LIN {X 0,Y 373.397,Z 455.176,A -85,B 0,C 180,E1 -12866.615,E2 -12866.615} C_VEL
LIN {X 0,Y 372.645,Z 466.782,A -85,B 0,C 180,E1 -12867.431,E2 -12867.431} C_VEL
LIN {X 0,Y 371.772,Z 478.488,A -85,B 0,C 180,E1 -12868.51,E2 -12868.51} C_VEL
LIN {X 0,Y 370.845,Z 489.006,A -85,B 0,C 180,E1 -12869.728,E2 -12869.728} C_VEL
LIN {X 0,Y 369.997,Z 498.484,A -85,B 0,C 180,E1 -12871.087,E2 -12871.087} C_VEL
LIN {X 0,Y 369.105,Z 507.613,A -85,B 0,C 180,E1 -12872.727,E2 -12872.727} C_VEL
LIN {X 0,Y 368.474,Z 514.962,A -85,B 0,C 180,E1 -12874.374,E2 -12874.374} C_VEL
LIN {X 0,Y 368.116,Z 520.845,A -85,B 0,C 180,E1 -12876.026,E2 -12876.026} C_VEL
LIN {X 0,Y 367.769,Z 525.5,A -85,B 0,C 180,E1 -12877.686,E2 -12877.686} C_VEL
LIN {X 0,Y 367.515,Z 529.046,A -85,B 0,C 180,E1 -12879.354,E2 -12879.354} C_VEL
LIN {X 0,Y 367.376,Z 531.568,A -85,B 0,C 180,E1 -12881.028,E2 -12881.028} C_VEL
LIN {X 0,Y 367.353,Z 533.088,A -85,B 0,C 180,E1 -12882.657,E2 -12882.657} C_VEL
LIN {X 0,Y 367.241,Z 533.754,A -85,B 0,C 180,E1 -12884.404,E2 -12884.404} C_VEL
LIN {X 0,Y 367.257,Z 533.671,A -85,B 0,C 180,E1 -12885.539,E2 -12885.539} C_VEL
LIN {X 0,Y 367.386,Z 532.771,A -85,B 0,C 180,E1 -12887.131,E2 -12887.131} C_VEL
LIN {X 0,Y 367.617,Z 530.783,A -85,B 0,C 180,E1 -12888.964,E2 -12888.964} C_VEL
LIN {X 0,Y 367.953,Z 527.938,A -85,B 0,C 180,E1 -12890.625,E2 -12890.625} C_VEL
LIN {X 0,Y 368.238,Z 525.407,A -85,B 0,C 180,E1 -12891.755,E2 -12891.755} C_VEL
LIN {X 0,Y 367.828,Z 523.313,A -85,B 0,C 180,E1 -12892.614,E2 -12892.614} C_VEL
LIN {X 0,Y 365.519,Z 519.519,A -85,B 0,C 180,E1 -12894.001,E2 -12894.001} C_VEL
LIN {X 0,Y 363.313,Z 515.047,A -85,B 0,C 180,E1 -12895.351,E2 -12895.351} C_VEL
LIN {X 0,Y 363.065,Z 511.888,A -85,B 0,C 180,E1 -12896.139,E2 -12896.139} C_VEL
LIN {X 0,Y 364.268,Z 503.365,A -85,B 0,C 180,E1 -12897.895,E2 -12897.895} C_VEL
LIN {X 0,Y 365.394,Z 494.439,A -85,B 0,C 180,E1 -12899.37,E2 -12899.37} C_VEL
LIN {X 0,Y 366.725,Z 483.898,A -85,B 0,C 180,E1 -12900.759,E2 -12900.759} C_VEL
LIN {X 0,Y 367.92,Z 473.579,A -85,B 0,C 180,E1 -12901.848,E2 -12901.848} C_VEL
LIN {X 0,Y 368.964,Z 462.928,A -85,B 0,C 180,E1 -12902.747,E2 -12902.747} C_VEL
LIN {X 0,Y 369.916,Z 451.086,A -85,B 0,C 180,E1 -12903.514,E2 -12903.514} C_VEL
LIN {X 0,Y 370.609,Z 438.576,A -85,B 0,C 180,E1 -12904.096,E2 -12904.096} C_VEL
LIN {X 0,Y 371.139,Z 424.92,A -85,B 0,C 180,E1 -12904.492,E2 -12904.492} C_VEL
LIN {X 0,Y 372.654,Z 349.861,A -85,B 0,C 180,E1 -12905.968,E2 -12905.968} C_VEL
LIN {X 0,Y 368.76,Z 332.715,A -85,B 0,C 180,E1 -12906.629,E2 -12906.629} C_VEL
LIN {X 0,Y 364.625,Z 322.839,A -85,B 0,C 180,E1 -12907.207,E2 -12907.207} C_VEL
LIN {X 0,Y 362.63,Z 313.77,A -85,B 0,C 180,E1 -12909.757,E2 -12909.757} C_VEL
LIN {X 0,Y 361.806,Z 310.419,A -85,B 0,C 180,E1 -12910.75,E2 -12910.75} C_VEL
LIN {X 0,Y 361.809,Z 310.418,A -85,B 0,C 180,E1 -12914.368,E2 -12914.368} C_VEL
LIN {X 0,Y 361.822,Z 310.407,A -85,B 0,C 180,E1 -12917.569,E2 -12917.569} C_VEL
LIN {X 0,Y 361.836,Z 310.414,A -85,B 0,C 180,E1 -12921.572,E2 -12921.572} C_VEL
LIN {X 0,Y 361.865,Z 310.406,A -85,B 0,C 180,E1 -12924.655,E2 -12924.655} C_VEL
LIN {X 0,Y 361.829,Z 310.412,A -85,B 0,C 180,E1 -12928.37,E2 -12928.37} C_VEL
LIN {X 0,Y 361.857,Z 310.404,A -85,B 0,C 180,E1 -12930.952,E2 -12930.952} C_VEL
LIN {X 0,Y 361.859,Z 310.405,A -85,B 0,C 180,E1 -12934.705,E2 -12934.705} C_VEL
LIN {X 0,Y 361.852,Z 310.407,A -85,B 0,C 180,E1 -12938.345,E2 -12938.345} C_VEL
LIN {X 0,Y 361.895,Z 310.399,A -85,B 0,C 180,E1 -12942.093,E2 -12942.093} C_VEL
LIN {X 0,Y 361.97,Z 310.388,A -85,B 0,C 180,E1 -12946.113,E2 -12946.113} C_VEL
LIN {X 0,Y 361.985,Z 310.393,A -85,B 0,C 180,E1 -12949.937,E2 -12949.937} C_VEL
LIN {X 0,Y 362.106,Z 310.375,A -85,B 0,C 180,E1 -12953.313,E2 -12953.313} C_VEL
LIN {X 0,Y 362.246,Z 310.353,A -85,B 0,C 180,E1 -12957.776,E2 -12957.776} C_VEL
LIN {X 0,Y 362.247,Z 310.351,A -85,B 0,C 180,E1 -12962.224,E2 -12962.224} C_VEL
LIN {X 0,Y 362.131,Z 310.368,A -85,B 0,C 180,E1 -12966.687,E2 -12966.687} C_VEL
LIN {X 0,Y 361.988,Z 310.389,A -85,B 0,C 180,E1 -12970.064,E2 -12970.064} C_VEL
LIN {X 0,Y 361.99,Z 310.382,A -85,B 0,C 180,E1 -12973.899,E2 -12973.899} C_VEL
LIN {X 0,Y 361.92,Z 310.396,A -85,B 0,C 180,E1 -12976.935,E2 -12976.935} C_VEL
LIN {X 0,Y 361.879,Z 310.403,A -85,B 0,C 180,E1 -12980.462,E2 -12980.462} C_VEL
LIN {X 0,Y 361.853,Z 310.405,A -85,B 0,C 180,E1 -12984.102,E2 -12984.102} C_VEL
LIN {X 0,Y 361.838,Z 310.406,A -85,B 0,C 180,E1 -12987.785,E2 -12987.785} C_VEL
LIN {X 0,Y 361.84,Z 310.408,A -85,B 0,C 180,E1 -12991.286,E2 -12991.286} C_VEL
LIN {X 0,Y 361.848,Z 310.409,A -85,B 0,C 180,E1 -12994.281,E2 -12994.281} C_VEL
LIN {X 0,Y 361.854,Z 310.411,A -85,B 0,C 180,E1 -12997.223,E2 -12997.223} C_VEL
LIN {X 0,Y 361.807,Z 310.416,A -85,B 0,C 180,E1 -13000.752,E2 -13000.752} C_VEL
LIN {X 0,Y 361.811,Z 310.405,A -85,B 0,C 180,E1 -13004.37,E2 -13004.37} C_VEL
LIN {X 0,Y 361.831,Z 310.415,A -85,B 0,C 180,E1 -13007.569,E2 -13007.569} C_VEL
LIN {X 0,Y 361.862,Z 310.412,A -85,B 0,C 180,E1 -13010.975,E2 -13010.975} C_VEL
LIN {X 0,Y 361.871,Z 310.406,A -85,B 0,C 180,E1 -13014.656,E2 -13014.656} C_VEL
LIN {X 0,Y 361.835,Z 310.411,A -85,B 0,C 180,E1 -13018.372,E2 -13018.372} C_VEL
LIN {X 0,Y 361.903,Z 310.527,A -85,B 0,C 180,E1 -13019.004,E2 -13019.004} C_VEL
LIN {X 0,Y 364.589,Z 321.736,A -85,B 0,C 180,E1 -13022.133,E2 -13022.133} C_VEL
LIN {X 0,Y 366.327,Z 331.239,A -85,B 0,C 180,E1 -13024.628,E2 -13024.628} C_VEL
LIN {X 0,Y 366.472,Z 334.158,A -85,B 0,C 180,E1 -13025.349,E2 -13025.349} C_VEL
LIN {X 0,Y 365.703,Z 341.412,A -85,B 0,C 180,E1 -13026.981,E2 -13026.981} C_VEL
LIN {X 0,Y 370.351,Z 363.93,A -85,B 0,C 180,E1 -13027.82,E2 -13027.82} C_VEL
LIN {X 0,Y 372.213,Z 375.715,A -85,B 0,C 180,E1 -13028.207,E2 -13028.207} C_VEL
LIN {X 0,Y 370.773,Z 449.685,A -85,B 0,C 180,E1 -13029.69,E2 -13029.69} C_VEL
LIN {X 0,Y 369.999,Z 462.791,A -85,B 0,C 180,E1 -13030.153,E2 -13030.153} C_VEL
LIN {X 0,Y 369.057,Z 475.405,A -85,B 0,C 180,E1 -13030.824,E2 -13030.824} C_VEL
LIN {X 0,Y 367.953,Z 486.664,A -85,B 0,C 180,E1 -13031.631,E2 -13031.631} C_VEL
LIN {X 0,Y 366.614,Z 498.29,A -85,B 0,C 180,E1 -13032.716,E2 -13032.716} C_VEL
LIN {X 0,Y 365.281,Z 508.754,A -85,B 0,C 180,E1 -13033.945,E2 -13033.945} C_VEL
LIN {X 0,Y 364.256,Z 517.807,A -85,B 0,C 180,E1 -13035.268,E2 -13035.268} C_VEL
LIN {X 0,Y 363.039,Z 526.654,A -85,B 0,C 180,E1 -13036.853,E2 -13036.853} C_VEL
LIN {X 0,Y 362.012,Z 534.145,A -85,B 0,C 180,E1 -13038.523,E2 -13038.523} C_VEL
LIN {X 0,Y 361.207,Z 541.091,A -85,B 0,C 180,E1 -13040.482,E2 -13040.482} C_VEL
LIN {X 0,Y 360.731,Z 545.697,A -85,B 0,C 180,E1 -13042.163,E2 -13042.163} C_VEL
LIN {X 0,Y 360.425,Z 549.441,A -85,B 0,C 180,E1 -13043.969,E2 -13043.969} C_VEL
LIN {X 0,Y 360.349,Z 551.741,A -85,B 0,C 180,E1 -13045.527,E2 -13045.527} C_VEL
LIN {X 0,Y 360.296,Z 552.926,A -85,B 0,C 180,E1 -13046.646,E2 -13046.646} C_VEL
LIN {X 0,Y 360.303,Z 554.036,A -85,B 0,C 180,E1 -13048.883,E2 -13048.883} C_VEL
LIN {X 0,Y 360.36,Z 554.014,A -85,B 0,C 180,E1 -13050.001,E2 -13050.001} C_VEL
LIN {X 0,Y 360.321,Z 553.599,A -85,B 0,C 180,E1 -13051.119,E2 -13051.119} C_VEL
LIN {X 0,Y 360.279,Z 552.743,A -85,B 0,C 180,E1 -13052.237,E2 -13052.237} C_VEL
LIN {X 0,Y 360.303,Z 551.485,A -85,B 0,C 180,E1 -13053.356,E2 -13053.356} C_VEL
LIN {X 0,Y 360.368,Z 548.805,A -85,B 0,C 180,E1 -13055.036,E2 -13055.036} C_VEL
LIN {X 0,Y 360.499,Z 545.09,A -85,B 0,C 180,E1 -13056.718,E2 -13056.718} C_VEL
LIN {X 0,Y 360.758,Z 540.241,A -85,B 0,C 180,E1 -13058.402,E2 -13058.402} C_VEL
LIN {X 0,Y 361.198,Z 534.109,A -85,B 0,C 180,E1 -13060.086,E2 -13060.086} C_VEL
LIN {X 0,Y 361.821,Z 526.469,A -85,B 0,C 180,E1 -13061.769,E2 -13061.769} C_VEL
LIN {X 0,Y 362.552,Z 518.648,A -85,B 0,C 180,E1 -13063.167,E2 -13063.167} C_VEL
LIN {X 0,Y 363.53,Z 508.156,A -85,B 0,C 180,E1 -13064.679,E2 -13064.679} C_VEL
LIN {X 0,Y 364.383,Z 497.129,A -85,B 0,C 180,E1 -13065.954,E2 -13065.954} C_VEL
LIN {X 0,Y 365.32,Z 486.561,A -85,B 0,C 180,E1 -13066.917,E2 -13066.917} C_VEL
LIN {X 0,Y 366.214,Z 473.802,A -85,B 0,C 180,E1 -13067.811,E2 -13067.811} C_VEL
LIN {X 0,Y 367.003,Z 461.06,A -85,B 0,C 180,E1 -13068.456,E2 -13068.456} C_VEL
LIN {X 0,Y 367.492,Z 448.899,A -85,B 0,C 180,E1 -13068.865,E2 -13068.865} C_VEL
LIN {X 0,Y 368.603,Z 374.28,A -85,B 0,C 180,E1 -13070.333,E2 -13070.333} C_VEL
LIN {X 0,Y 363.878,Z 341.672,A -85,B 0,C 180,E1 -13071.223,E2 -13071.223} C_VEL
LIN {X 0,Y 364.97,Z 328.754,A -85,B 0,C 180,E1 -13074.155,E2 -13074.155} C_VEL
LIN {X 0,Y 364.684,Z 324.827,A -85,B 0,C 180,E1 -13075.087,E2 -13075.087} C_VEL
LIN {X 0,Y 362.4,Z 312.879,A -85,B 0,C 180,E1 -13078.053,E2 -13078.053} C_VEL
LIN {X 0,Y 361.927,Z 310.4,A -85,B 0,C 180,E1 -13078.726,E2 -13078.726} C_VEL
LIN {X 0,Y 361.842,Z 310.412,A -85,B 0,C 180,E1 -13081.63,E2 -13081.63} C_VEL
LIN {X 0,Y 361.879,Z 310.404,A -85,B 0,C 180,E1 -13085.345,E2 -13085.345} C_VEL
LIN {X 0,Y 361.83,Z 310.41,A -85,B 0,C 180,E1 -13089.018,E2 -13089.018} C_VEL
LIN {X 0,Y 361.837,Z 310.41,A -85,B 0,C 180,E1 -13092.83,E2 -13092.83} C_VEL
LIN {X 0,Y 361.822,Z 310.413,A -85,B 0,C 180,E1 -13095.947,E2 -13095.947} C_VEL
LIN {X 0,Y 361.835,Z 310.41,A -85,B 0,C 180,E1 -13099.246,E2 -13099.246} C_VEL
LIN {X 0,Y 361.867,Z 310.411,A -85,B 0,C 180,E1 -13102.778,E2 -13102.778} C_VEL
LIN {X 0,Y 361.859,Z 310.406,A -85,B 0,C 180,E1 -13105.72,E2 -13105.72} C_VEL
LIN {X 0,Y 361.871,Z 310.405,A -85,B 0,C 180,E1 -13109.671,E2 -13109.671} C_VEL
LIN {X 0,Y 361.905,Z 310.403,A -85,B 0,C 180,E1 -13113.471,E2 -13113.471} C_VEL
LIN {X 0,Y 361.882,Z 310.409,A -85,B 0,C 180,E1 -13117.144,E2 -13117.144} C_VEL
LIN {X 0,Y 361.89,Z 310.403,A -85,B 0,C 180,E1 -13120.722,E2 -13120.722} C_VEL
LIN {X 0,Y 361.948,Z 310.395,A -85,B 0,C 180,E1 -13124.226,E2 -13124.226} C_VEL
LIN {X 0,Y 362.003,Z 310.388,A -85,B 0,C 180,E1 -13126.528,E2 -13126.528} C_VEL
LIN {X 0,Y 362.032,Z 310.389,A -85,B 0,C 180,E1 -13129.938,E2 -13129.938} C_VEL
LIN {X 0,Y 362.15,Z 310.371,A -85,B 0,C 180,E1 -13133.313,E2 -13133.313} C_VEL
LIN {X 0,Y 362.274,Z 310.358,A -85,B 0,C 180,E1 -13137.776,E2 -13137.776} C_VEL
LIN {X 0,Y 362.405,Z 310.344,A -85,B 0,C 180,E1 -13140,E2 -13140} C_VEL
LIN {X 0,Y 362.275,Z 310.361,A -85,B 0,C 180,E1 -13142.223,E2 -13142.223} C_VEL
LIN {X 0,Y 362.127,Z 310.376,A -85,B 0,C 180,E1 -13146.687,E2 -13146.687} C_VEL
LIN {X 0,Y 362.003,Z 310.39,A -85,B 0,C 180,E1 -13150.063,E2 -13150.063} C_VEL
LIN {X 0,Y 362.002,Z 310.389,A -85,B 0,C 180,E1 -13153.898,E2 -13153.898} C_VEL
LIN {X 0,Y 361.932,Z 310.402,A -85,B 0,C 180,E1 -13156.934,E2 -13156.934} C_VEL
LIN {X 0,Y 361.89,Z 310.405,A -85,B 0,C 180,E1 -13160.46,E2 -13160.46} C_VEL
LIN {X 0,Y 361.896,Z 310.401,A -85,B 0,C 180,E1 -13164.112,E2 -13164.112} C_VEL
LIN {X 0,Y 361.867,Z 310.406,A -85,B 0,C 180,E1 -13167.782,E2 -13167.782} C_VEL
LIN {X 0,Y 361.85,Z 310.414,A -85,B 0,C 180,E1 -13171.285,E2 -13171.285} C_VEL
LIN {X 0,Y 361.857,Z 310.406,A -85,B 0,C 180,E1 -13174.28,E2 -13174.28} C_VEL
LIN {X 0,Y 361.871,Z 310.408,A -85,B 0,C 180,E1 -13177.223,E2 -13177.223} C_VEL
LIN {X 0,Y 361.832,Z 310.409,A -85,B 0,C 180,E1 -13180.754,E2 -13180.754} C_VEL
LIN {X 0,Y 361.819,Z 310.412,A -85,B 0,C 180,E1 -13184.368,E2 -13184.368} C_VEL
LIN {X 0,Y 361.834,Z 310.412,A -85,B 0,C 180,E1 -13187.568,E2 -13187.568} C_VEL
LIN {X 0,Y 361.832,Z 310.409,A -85,B 0,C 180,E1 -13190.98,E2 -13190.98} C_VEL
LIN {X 0,Y 361.876,Z 310.406,A -85,B 0,C 180,E1 -13194.655,E2 -13194.655} C_VEL
LIN {X 0,Y 361.839,Z 310.415,A -85,B 0,C 180,E1 -13198.37,E2 -13198.37} C_VEL
LIN {X 0,Y 361.867,Z 310.407,A -85,B 0,C 180,E1 -13200.951,E2 -13200.951} C_VEL
LIN {X 0,Y 361.905,Z 310.406,A -85,B 0,C 180,E1 -13204.707,E2 -13204.707} C_VEL
LIN {X 0,Y 361.892,Z 310.405,A -85,B 0,C 180,E1 -13208.346,E2 -13208.346} C_VEL
LIN {X 0,Y 361.921,Z 310.399,A -85,B 0,C 180,E1 -13212.084,E2 -13212.084} C_VEL
LIN {X 0,Y 361.963,Z 310.396,A -85,B 0,C 180,E1 -13215.379,E2 -13215.379} C_VEL
LIN {X 0,Y 361.97,Z 310.395,A -85,B 0,C 180,E1 -13218.803,E2 -13218.803} C_VEL
LIN {X 0,Y 362.024,Z 310.399,A -85,B 0,C 180,E1 -13219.584,E2 -13219.584} C_VEL
LIN {X 0,Y 364.038,Z 321.449,A -85,B 0,C 180,E1 -13222.511,E2 -13222.511} C_VEL
LIN {X 0,Y 364.025,Z 322.81,A -85,B 0,C 180,E1 -13222.853,E2 -13222.853} C_VEL
LIN {X 0,Y 368.879,Z 348.378,A -85,B 0,C 180,E1 -13223.613,E2 -13223.613} C_VEL
LIN {X 0,Y 367.57,Z 430.446,A -85,B 0,C 180,E1 -13225.235,E2 -13225.235} C_VEL
LIN {X 0,Y 367.096,Z 442.918,A -85,B 0,C 180,E1 -13225.682,E2 -13225.682} C_VEL
LIN {X 0,Y 366.522,Z 455.189,A -85,B 0,C 180,E1 -13226.334,E2 -13226.334} C_VEL
LIN {X 0,Y 365.706,Z 467.767,A -85,B 0,C 180,E1 -13227.245,E2 -13227.245} C_VEL
LIN {X 0,Y 364.788,Z 479.321,A -85,B 0,C 180,E1 -13228.343,E2 -13228.343} C_VEL
LIN {X 0,Y 363.84,Z 489.73,A -85,B 0,C 180,E1 -13229.584,E2 -13229.584} C_VEL
LIN {X 0,Y 363.022,Z 498.243,A -85,B 0,C 180,E1 -13230.831,E2 -13230.831} C_VEL
LIN {X 0,Y 362.239,Z 506.097,A -85,B 0,C 180,E1 -13232.223,E2 -13232.223} C_VEL
LIN {X 0,Y 361.573,Z 513.752,A -85,B 0,C 180,E1 -13233.9,E2 -13233.9} C_VEL
LIN {X 0,Y 361.101,Z 519.906,A -85,B 0,C 180,E1 -13235.583,E2 -13235.583} C_VEL
LIN {X 0,Y 360.767,Z 524.795,A -85,B 0,C 180,E1 -13237.274,E2 -13237.274} C_VEL
LIN {X 0,Y 360.486,Z 528.566,A -85,B 0,C 180,E1 -13238.972,E2 -13238.972} C_VEL
LIN {X 0,Y 360.315,Z 530.517,A -85,B 0,C 180,E1 -13240.109,E2 -13240.109} C_VEL
LIN {X 0,Y 360.277,Z 532.016,A -85,B 0,C 180,E1 -13241.248,E2 -13241.248} C_VEL
LIN {X 0,Y 360.255,Z 533.312,A -85,B 0,C 180,E1 -13242.731,E2 -13242.731} C_VEL
LIN {X 0,Y 360.164,Z 533.985,A -85,B 0,C 180,E1 -13244.694,E2 -13244.694} C_VEL
LIN {X 0,Y 360.193,Z 533.788,A -85,B 0,C 180,E1 -13245.851,E2 -13245.851} C_VEL
LIN {X 0,Y 360.294,Z 533.113,A -85,B 0,C 180,E1 -13247.098,E2 -13247.098} C_VEL
LIN {X 0,Y 360.431,Z 532.147,A -85,B 0,C 180,E1 -13248.178,E2 -13248.178} C_VEL
LIN {X 0,Y 360.587,Z 530.668,A -85,B 0,C 180,E1 -13249.349,E2 -13249.349} C_VEL
LIN {X 0,Y 360.936,Z 528.118,A -85,B 0,C 180,E1 -13250.831,E2 -13250.831} C_VEL
LIN {X 0,Y 361.521,Z 523.286,A -85,B 0,C 180,E1 -13252.879,E2 -13252.879} C_VEL
LIN {X 0,Y 362.27,Z 517.717,A -85,B 0,C 180,E1 -13254.65,E2 -13254.65} C_VEL
LIN {X 0,Y 363.065,Z 511.888,A -85,B 0,C 180,E1 -13256.139,E2 -13256.139} C_VEL
LIN {X 0,Y 362.853,Z 508.576,A -85,B 0,C 180,E1 -13256.909,E2 -13256.909} C_VEL
LIN {X 0,Y 360.873,Z 502.948,A -85,B 0,C 180,E1 -13258.166,E2 -13258.166} C_VEL
LIN {X 0,Y 359.004,Z 496.806,A -85,B 0,C 180,E1 -13259.365,E2 -13259.365} C_VEL
LIN {X 0,Y 358.954,Z 492.621,A -85,B 0,C 180,E1 -13260.032,E2 -13260.032} C_VEL
LIN {X 0,Y 360.348,Z 481.906,A -85,B 0,C 180,E1 -13261.413,E2 -13261.413} C_VEL
LIN {X 0,Y 361.754,Z 469.821,A -85,B 0,C 180,E1 -13262.622,E2 -13262.622} C_VEL
LIN {X 0,Y 362.906,Z 457.64,A -85,B 0,C 180,E1 -13263.564,E2 -13263.564} C_VEL
LIN {X 0,Y 363.787,Z 444.948,A -85,B 0,C 180,E1 -13264.281,E2 -13264.281} C_VEL
LIN {X 0,Y 364.474,Z 431.327,A -85,B 0,C 180,E1 -13264.794,E2 -13264.794} C_VEL
LIN {X 0,Y 366.244,Z 350.87,A -85,B 0,C 180,E1 -13266.432,E2 -13266.432} C_VEL
LIN {X 0,Y 362.63,Z 335.151,A -85,B 0,C 180,E1 -13267.063,E2 -13267.063} C_VEL
LIN {X 0,Y 357.555,Z 323.096,A -85,B 0,C 180,E1 -13267.779,E2 -13267.779} C_VEL
LIN {X 0,Y 355.144,Z 312.821,A -85,B 0,C 180,E1 -13270.77,E2 -13270.77} C_VEL
LIN {X 0,Y 354.776,Z 311.29,A -85,B 0,C 180,E1 -13271.267,E2 -13271.267} C_VEL
LIN {X 0,Y 354.756,Z 311.297,A -85,B 0,C 180,E1 -13274.505,E2 -13274.505} C_VEL
LIN {X 0,Y 354.781,Z 311.285,A -85,B 0,C 180,E1 -13277.661,E2 -13277.661} C_VEL
LIN {X 0,Y 354.777,Z 311.292,A -85,B 0,C 180,E1 -13280.661,E2 -13280.661} C_VEL
LIN {X 0,Y 354.813,Z 311.287,A -85,B 0,C 180,E1 -13284.3,E2 -13284.3} C_VEL
LIN {X 0,Y 354.778,Z 311.284,A -85,B 0,C 180,E1 -13287.666,E2 -13287.666} C_VEL
LIN {X 0,Y 354.793,Z 311.289,A -85,B 0,C 180,E1 -13291.614,E2 -13291.614} C_VEL
LIN {X 0,Y 354.797,Z 311.288,A -85,B 0,C 180,E1 -13295.419,E2 -13295.419} C_VEL
LIN {X 0,Y 354.815,Z 311.284,A -85,B 0,C 180,E1 -13299.113,E2 -13299.113} C_VEL
LIN {X 0,Y 354.842,Z 311.278,A -85,B 0,C 180,E1 -13302.717,E2 -13302.717} C_VEL
LIN {X 0,Y 354.93,Z 311.263,A -85,B 0,C 180,E1 -13306.255,E2 -13306.255} C_VEL
LIN {X 0,Y 354.941,Z 311.271,A -85,B 0,C 180,E1 -13309.735,E2 -13309.735} C_VEL
LIN {X 0,Y 355.073,Z 311.251,A -85,B 0,C 180,E1 -13313.18,E2 -13313.18} C_VEL
LIN {X 0,Y 355.208,Z 311.229,A -85,B 0,C 180,E1 -13317.732,E2 -13317.732} C_VEL
LIN {X 0,Y 355.161,Z 311.236,A -85,B 0,C 180,E1 -13321.134,E2 -13321.134} C_VEL
LIN {X 0,Y 355.209,Z 311.227,A -85,B 0,C 180,E1 -13322.268,E2 -13322.268} C_VEL
LIN {X 0,Y 355.094,Z 311.243,A -85,B 0,C 180,E1 -13326.82,E2 -13326.82} C_VEL
LIN {X 0,Y 354.945,Z 311.268,A -85,B 0,C 180,E1 -13330.265,E2 -13330.265} C_VEL
LIN {X 0,Y 354.935,Z 311.261,A -85,B 0,C 180,E1 -13334.019,E2 -13334.019} C_VEL
LIN {X 0,Y 354.882,Z 311.265,A -85,B 0,C 180,E1 -13338.093,E2 -13338.093} C_VEL
LIN {X 0,Y 354.811,Z 311.284,A -85,B 0,C 180,E1 -13341.418,E2 -13341.418} C_VEL
LIN {X 0,Y 354.797,Z 311.285,A -85,B 0,C 180,E1 -13344.581,E2 -13344.581} C_VEL
LIN {X 0,Y 354.794,Z 311.284,A -85,B 0,C 180,E1 -13348.386,E2 -13348.386} C_VEL
LIN {X 0,Y 354.78,Z 311.287,A -85,B 0,C 180,E1 -13352.334,E2 -13352.334} C_VEL
LIN {X 0,Y 354.816,Z 311.283,A -85,B 0,C 180,E1 -13355.7,E2 -13355.7} C_VEL
LIN {X 0,Y 354.762,Z 311.29,A -85,B 0,C 180,E1 -13359.414,E2 -13359.414} C_VEL
LIN {X 0,Y 354.78,Z 311.277,A -85,B 0,C 180,E1 -13362.868,E2 -13362.868} C_VEL
LIN {X 0,Y 354.763,Z 311.299,A -85,B 0,C 180,E1 -13366.105,E2 -13366.105} C_VEL
LIN {X 0,Y 354.782,Z 311.295,A -85,B 0,C 180,E1 -13369.18,E2 -13369.18} C_VEL
LIN {X 0,Y 354.803,Z 311.292,A -85,B 0,C 180,E1 -13372.404,E2 -13372.404} C_VEL
LIN {X 0,Y 354.809,Z 311.284,A -85,B 0,C 180,E1 -13374.942,E2 -13374.942} C_VEL
LIN {X 0,Y 354.826,Z 311.36,A -85,B 0,C 180,E1 -13378.485,E2 -13378.485} C_VEL
LIN {X 0,Y 357.668,Z 323.152,A -85,B 0,C 180,E1 -13381.864,E2 -13381.864} C_VEL
LIN {X 0,Y 359.521,Z 333.07,A -85,B 0,C 180,E1 -13384.53,E2 -13384.53} C_VEL
LIN {X 0,Y 359.451,Z 336.813,A -85,B 0,C 180,E1 -13385.452,E2 -13385.452} C_VEL
LIN {X 0,Y 358.954,Z 340.866,A -85,B 0,C 180,E1 -13386.41,E2 -13386.41} C_VEL
LIN {X 0,Y 363.737,Z 363.679,A -85,B 0,C 180,E1 -13387.311,E2 -13387.311} C_VEL
LIN {X 0,Y 365.805,Z 376.443,A -85,B 0,C 180,E1 -13387.748,E2 -13387.748} C_VEL
LIN {X 0,Y 364.295,Z 449.545,A -85,B 0,C 180,E1 -13389.239,E2 -13389.239} C_VEL
LIN {X 0,Y 363.485,Z 462.632,A -85,B 0,C 180,E1 -13389.708,E2 -13389.708} C_VEL
LIN {X 0,Y 362.514,Z 475.234,A -85,B 0,C 180,E1 -13390.39,E2 -13390.39} C_VEL
LIN {X 0,Y 361.256,Z 487.279,A -85,B 0,C 180,E1 -13391.278,E2 -13391.278} C_VEL
LIN {X 0,Y 359.855,Z 498.75,A -85,B 0,C 180,E1 -13392.38,E2 -13392.38} C_VEL
LIN {X 0,Y 358.479,Z 509.1,A -85,B 0,C 180,E1 -13393.632,E2 -13393.632} C_VEL
LIN {X 0,Y 357.377,Z 518.197,A -85,B 0,C 180,E1 -13395.001,E2 -13395.001} C_VEL
LIN {X 0,Y 356.113,Z 526.8,A -85,B 0,C 180,E1 -13396.593,E2 -13396.593} C_VEL
LIN {X 0,Y 355.036,Z 534.224,A -85,B 0,C 180,E1 -13398.294,E2 -13398.294} C_VEL
LIN {X 0,Y 354.171,Z 541.102,A -85,B 0,C 180,E1 -13400.291,E2 -13400.291} C_VEL
LIN {X 0,Y 353.691,Z 545.658,A -85,B 0,C 180,E1 -13402.006,E2 -13402.006} C_VEL
LIN {X 0,Y 353.352,Z 549.554,A -85,B 0,C 180,E1 -13403.978,E2 -13403.978} C_VEL
LIN {X 0,Y 353.264,Z 551.627,A -85,B 0,C 180,E1 -13405.437,E2 -13405.437} C_VEL
LIN {X 0,Y 353.218,Z 552.776,A -85,B 0,C 180,E1 -13406.579,E2 -13406.579} C_VEL
LIN {X 0,Y 353.203,Z 553.846,A -85,B 0,C 180,E1 -13408.861,E2 -13408.861} C_VEL
LIN {X 0,Y 353.262,Z 553.805,A -85,B 0,C 180,E1 -13410.001,E2 -13410.001} C_VEL
LIN {X 0,Y 353.222,Z 553.359,A -85,B 0,C 180,E1 -13411.141,E2 -13411.141} C_VEL
LIN {X 0,Y 353.225,Z 551.201,A -85,B 0,C 180,E1 -13413.423,E2 -13413.423} C_VEL
LIN {X 0,Y 353.27,Z 548.479,A -85,B 0,C 180,E1 -13415.137,E2 -13415.137} C_VEL
LIN {X 0,Y 353.416,Z 544.721,A -85,B 0,C 180,E1 -13416.854,E2 -13416.854} C_VEL
LIN {X 0,Y 353.698,Z 539.825,A -85,B 0,C 180,E1 -13418.571,E2 -13418.571} C_VEL
LIN {X 0,Y 354.168,Z 533.641,A -85,B 0,C 180,E1 -13420.289,E2 -13420.289} C_VEL
LIN {X 0,Y 354.844,Z 525.936,A -85,B 0,C 180,E1 -13422.004,E2 -13422.004} C_VEL
LIN {X 0,Y 355.57,Z 518.028,A -85,B 0,C 180,E1 -13423.43,E2 -13423.43} C_VEL
LIN {X 0,Y 356.537,Z 508.362,A -85,B 0,C 180,E1 -13424.849,E2 -13424.849} C_VEL
LIN {X 0,Y 357.385,Z 497.599,A -85,B 0,C 180,E1 -13426.128,E2 -13426.128} C_VEL
LIN {X 0,Y 358.334,Z 487.208,A -85,B 0,C 180,E1 -13427.11,E2 -13427.11} C_VEL
LIN {X 0,Y 359.28,Z 474.758,A -85,B 0,C 180,E1 -13428.019,E2 -13428.019} C_VEL
LIN {X 0,Y 360.121,Z 461.64,A -85,B 0,C 180,E1 -13428.712,E2 -13428.712} C_VEL
LIN {X 0,Y 360.657,Z 448.707,A -85,B 0,C 180,E1 -13429.162,E2 -13429.162} C_VEL
LIN {X 0,Y 361.719,Z 374.275,A -85,B 0,C 180,E1 -13430.657,E2 -13430.657} C_VEL
LIN {X 0,Y 356.967,Z 341.403,A -85,B 0,C 180,E1 -13431.592,E2 -13431.592} C_VEL
LIN {X 0,Y 358.02,Z 329.505,A -85,B 0,C 180,E1 -13434.346,E2 -13434.346} C_VEL
LIN {X 0,Y 357.597,Z 325.585,A -85,B 0,C 180,E1 -13435.303,E2 -13435.303} C_VEL
LIN {X 0,Y 355.566,Z 314.707,A -85,B 0,C 180,E1 -13438.053,E2 -13438.053} C_VEL
LIN {X 0,Y 354.877,Z 311.278,A -85,B 0,C 180,E1 -13438.992,E2 -13438.992} C_VEL
LIN {X 0,Y 354.792,Z 311.289,A -85,B 0,C 180,E1 -13442.334,E2 -13442.334} C_VEL
LIN {X 0,Y 354.826,Z 311.285,A -85,B 0,C 180,E1 -13445.7,E2 -13445.7} C_VEL
LIN {X 0,Y 354.772,Z 311.289,A -85,B 0,C 180,E1 -13449.413,E2 -13449.413} C_VEL
LIN {X 0,Y 354.79,Z 311.288,A -85,B 0,C 180,E1 -13452.867,E2 -13452.867} C_VEL
LIN {X 0,Y 354.771,Z 311.292,A -85,B 0,C 180,E1 -13456.104,E2 -13456.104} C_VEL
LIN {X 0,Y 354.787,Z 311.288,A -85,B 0,C 180,E1 -13459.179,E2 -13459.179} C_VEL
LIN {X 0,Y 354.81,Z 311.288,A -85,B 0,C 180,E1 -13462.403,E2 -13462.403} C_VEL
LIN {X 0,Y 354.816,Z 311.288,A -85,B 0,C 180,E1 -13464.941,E2 -13464.941} C_VEL
LIN {X 0,Y 354.798,Z 311.288,A -85,B 0,C 180,E1 -13468.405,E2 -13468.405} C_VEL
LIN {X 0,Y 354.814,Z 311.285,A -85,B 0,C 180,E1 -13471.616,E2 -13471.616} C_VEL
LIN {X 0,Y 354.858,Z 311.282,A -85,B 0,C 180,E1 -13475.423,E2 -13475.423} C_VEL
LIN {X 0,Y 354.831,Z 311.286,A -85,B 0,C 180,E1 -13479.113,E2 -13479.113} C_VEL
LIN {X 0,Y 354.885,Z 311.275,A -85,B 0,C 180,E1 -13482.719,E2 -13482.719} C_VEL
LIN {X 0,Y 354.956,Z 311.267,A -85,B 0,C 180,E1 -13486.255,E2 -13486.255} C_VEL
LIN {X 0,Y 354.979,Z 311.27,A -85,B 0,C 180,E1 -13489.736,E2 -13489.736} C_VEL
LIN {X 0,Y 355.114,Z 311.247,A -85,B 0,C 180,E1 -13493.18,E2 -13493.18} C_VEL
LIN {X 0,Y 355.236,Z 311.235,A -85,B 0,C 180,E1 -13497.732,E2 -13497.732} C_VEL
LIN {X 0,Y 355.355,Z 311.222,A -85,B 0,C 180,E1 -13500,E2 -13500} C_VEL
LIN {X 0,Y 355.238,Z 311.237,A -85,B 0,C 180,E1 -13502.267,E2 -13502.267} C_VEL
LIN {X 0,Y 355.092,Z 311.251,A -85,B 0,C 180,E1 -13506.82,E2 -13506.82} C_VEL
LIN {X 0,Y 354.959,Z 311.27,A -85,B 0,C 180,E1 -13510.264,E2 -13510.264} C_VEL
LIN {X 0,Y 354.946,Z 311.268,A -85,B 0,C 180,E1 -13514.018,E2 -13514.018} C_VEL
LIN {X 0,Y 354.893,Z 311.274,A -85,B 0,C 180,E1 -13518.092,E2 -13518.092} C_VEL
LIN {X 0,Y 354.818,Z 311.283,A -85,B 0,C 180,E1 -13522.107,E2 -13522.107} C_VEL
LIN {X 0,Y 354.866,Z 311.278,A -85,B 0,C 180,E1 -13525.83,E2 -13525.83} C_VEL
LIN {X 0,Y 354.81,Z 311.286,A -85,B 0,C 180,E1 -13529.682,E2 -13529.682} C_VEL
LIN {X 0,Y 354.817,Z 311.287,A -85,B 0,C 180,E1 -13533.683,E2 -13533.683} C_VEL
LIN {X 0,Y 354.801,Z 311.285,A -85,B 0,C 180,E1 -13536.459,E2 -13536.459} C_VEL
LIN {X 0,Y 354.827,Z 311.287,A -85,B 0,C 180,E1 -13539.423,E2 -13539.423} C_VEL
LIN {X 0,Y 354.788,Z 311.287,A -85,B 0,C 180,E1 -13542.866,E2 -13542.866} C_VEL
LIN {X 0,Y 354.769,Z 311.294,A -85,B 0,C 180,E1 -13546.103,E2 -13546.103} C_VEL
LIN {X 0,Y 354.784,Z 311.288,A -85,B 0,C 180,E1 -13549.177,E2 -13549.177} C_VEL
LIN {X 0,Y 354.803,Z 311.289,A -85,B 0,C 180,E1 -13552.403,E2 -13552.403} C_VEL
LIN {X 0,Y 354.813,Z 311.284,A -85,B 0,C 180,E1 -13554.94,E2 -13554.94} C_VEL
LIN {X 0,Y 354.795,Z 311.292,A -85,B 0,C 180,E1 -13558.404,E2 -13558.404} C_VEL
LIN {X 0,Y 354.811,Z 311.284,A -85,B 0,C 180,E1 -13561.615,E2 -13561.615} C_VEL
LIN {X 0,Y 354.855,Z 311.279,A -85,B 0,C 180,E1 -13565.422,E2 -13565.422} C_VEL
LIN {X 0,Y 354.841,Z 311.283,A -85,B 0,C 180,E1 -13569.113,E2 -13569.113} C_VEL
LIN {X 0,Y 354.881,Z 311.28,A -85,B 0,C 180,E1 -13572.718,E2 -13572.718} C_VEL
LIN {X 0,Y 354.952,Z 311.267,A -85,B 0,C 180,E1 -13576.254,E2 -13576.254} C_VEL
LIN {X 0,Y 354.992,Z 311.407,A -85,B 0,C 180,E1 -13579.375,E2 -13579.375} C_VEL
LIN {X 0,Y 356.856,Z 321.391,A -85,B 0,C 180,E1 -13582.075,E2 -13582.075} C_VEL
LIN {X 0,Y 357.139,Z 323.255,A -85,B 0,C 180,E1 -13582.512,E2 -13582.512} C_VEL
LIN {X 0,Y 362.125,Z 349.592,A -85,B 0,C 180,E1 -13583.312,E2 -13583.312} C_VEL
LIN {X 0,Y 360.736,Z 430.467,A -85,B 0,C 180,E1 -13584.934,E2 -13584.934} C_VEL
LIN {X 0,Y 360.27,Z 442.852,A -85,B 0,C 180,E1 -13585.384,E2 -13585.384} C_VEL
LIN {X 0,Y 359.679,Z 454.867,A -85,B 0,C 180,E1 -13586.027,E2 -13586.027} C_VEL
LIN {X 0,Y 358.883,Z 467.097,A -85,B 0,C 180,E1 -13586.911,E2 -13586.911} C_VEL
LIN {X 0,Y 357.923,Z 478.835,A -85,B 0,C 180,E1 -13588.03,E2 -13588.03} C_VEL
LIN {X 0,Y 356.956,Z 489.361,A -85,B 0,C 180,E1 -13589.294,E2 -13589.294} C_VEL
LIN {X 0,Y 356.062,Z 497.98,A -85,B 0,C 180,E1 -13590.564,E2 -13590.564} C_VEL
LIN {X 0,Y 355.255,Z 505.916,A -85,B 0,C 180,E1 -13591.983,E2 -13591.983} C_VEL
LIN {X 0,Y 354.583,Z 513.66,A -85,B 0,C 180,E1 -13593.692,E2 -13593.692} C_VEL
LIN {X 0,Y 354.054,Z 518.967,A -85,B 0,C 180,E1 -13595.124,E2 -13595.124} C_VEL
LIN {X 0,Y 353.764,Z 524.091,A -85,B 0,C 180,E1 -13596.845,E2 -13596.845} C_VEL
LIN {X 0,Y 353.45,Z 528.087,A -85,B 0,C 180,E1 -13598.575,E2 -13598.575} C_VEL
LIN {X 0,Y 353.202,Z 531.039,A -85,B 0,C 180,E1 -13600.315,E2 -13600.315} C_VEL
LIN {X 0,Y 353.164,Z 532.431,A -85,B 0,C 180,E1 -13601.477,E2 -13601.477} C_VEL
LIN {X 0,Y 353.153,Z 533.535,A -85,B 0,C 180,E1 -13602.805,E2 -13602.805} C_VEL
LIN {X 0,Y 353.117,Z 534.018,A -85,B 0,C 180,E1 -13603.817,E2 -13603.817} C_VEL
LIN {X 0,Y 353.062,Z 534.171,A -85,B 0,C 180,E1 -13604.996,E2 -13604.996} C_VEL
LIN {X 0,Y 353.212,Z 533.305,A -85,B 0,C 180,E1 -13607.24,E2 -13607.24} C_VEL
LIN {X 0,Y 353.376,Z 532.116,A -85,B 0,C 180,E1 -13608.553,E2 -13608.553} C_VEL
LIN {X 0,Y 353.729,Z 529.59,A -85,B 0,C 180,E1 -13610.345,E2 -13610.345} C_VEL
LIN {X 0,Y 354.201,Z 525.967,A -85,B 0,C 180,E1 -13612.146,E2 -13612.146} C_VEL
LIN {X 0,Y 354.877,Z 521.302,A -85,B 0,C 180,E1 -13613.893,E2 -13613.893} C_VEL
LIN {X 0,Y 355.786,Z 514.897,A -85,B 0,C 180,E1 -13615.757,E2 -13615.757} C_VEL
LIN {X 0,Y 356.75,Z 508.259,A -85,B 0,C 180,E1 -13617.306,E2 -13617.306} C_VEL
LIN {X 0,Y 358.091,Z 498.927,A -85,B 0,C 180,E1 -13619.06,E2 -13619.06} C_VEL
LIN {X 0,Y 358.954,Z 492.621,A -85,B 0,C 180,E1 -13620.032,E2 -13620.032} C_VEL
LIN {X 0,Y 358.914,Z 488.275,A -85,B 0,C 180,E1 -13620.673,E2 -13620.673} C_VEL
LIN {X 0,Y 357.14,Z 481.055,A -85,B 0,C 180,E1 -13621.727,E2 -13621.727} C_VEL
LIN {X 0,Y 355.399,Z 473.445,A -85,B 0,C 180,E1 -13622.7,E2 -13622.7} C_VEL
LIN {X 0,Y 355.379,Z 468.411,A -85,B 0,C 180,E1 -13623.2,E2 -13623.2} C_VEL
LIN {X 0,Y 356.433,Z 457.53,A -85,B 0,C 180,E1 -13624.036,E2 -13624.036} C_VEL
LIN {X 0,Y 357.369,Z 444.569,A -85,B 0,C 180,E1 -13624.77,E2 -13624.77} C_VEL
LIN {X 0,Y 358.031,Z 431.878,A -85,B 0,C 180,E1 -13625.255,E2 -13625.255} C_VEL
LIN {X 0,Y 359.547,Z 369.889,A -85,B 0,C 180,E1 -13626.545,E2 -13626.545} C_VEL
LIN {X 0,Y 359.893,Z 352.228,A -85,B 0,C 180,E1 -13626.908,E2 -13626.908} C_VEL
LIN {X 0,Y 356.76,Z 338.109,A -85,B 0,C 180,E1 -13627.481,E2 -13627.481} C_VEL
LIN {X 0,Y 350.38,Z 323.354,A -85,B 0,C 180,E1 -13628.389,E2 -13628.389} C_VEL
LIN {X 0,Y 348.109,Z 313.871,A -85,B 0,C 180,E1 -13631.233,E2 -13631.233} C_VEL
LIN {X 0,Y 347.74,Z 312.165,A -85,B 0,C 180,E1 -13631.789,E2 -13631.789} C_VEL
LIN {X 0,Y 347.698,Z 312.175,A -85,B 0,C 180,E1 -13635.026,E2 -13635.026} C_VEL
LIN {X 0,Y 347.734,Z 312.168,A -85,B 0,C 180,E1 -13638.398,E2 -13638.398} C_VEL
LIN {X 0,Y 347.749,Z 312.166,A -85,B 0,C 180,E1 -13642.678,E2 -13642.678} C_VEL
LIN {X 0,Y 347.74,Z 312.148,A -85,B 0,C 180,E1 -13645.956,E2 -13645.956} C_VEL
LIN {X 0,Y 347.73,Z 312.169,A -85,B 0,C 180,E1 -13649.651,E2 -13649.651} C_VEL
LIN {X 0,Y 347.737,Z 312.165,A -85,B 0,C 180,E1 -13653.6,E2 -13653.6} C_VEL
LIN {X 0,Y 347.743,Z 312.168,A -85,B 0,C 180,E1 -13656.159,E2 -13656.159} C_VEL
LIN {X 0,Y 347.768,Z 312.168,A -85,B 0,C 180,E1 -13659.907,E2 -13659.907} C_VEL
LIN {X 0,Y 347.788,Z 312.159,A -85,B 0,C 180,E1 -13663.566,E2 -13663.566} C_VEL
LIN {X 0,Y 347.875,Z 312.141,A -85,B 0,C 180,E1 -13667.16,E2 -13667.16} C_VEL
LIN {X 0,Y 347.924,Z 312.135,A -85,B 0,C 180,E1 -13670.701,E2 -13670.701} C_VEL
LIN {X 0,Y 348.024,Z 312.135,A -85,B 0,C 180,E1 -13674.205,E2 -13674.205} C_VEL
LIN {X 0,Y 348.145,Z 312.108,A -85,B 0,C 180,E1 -13677.686,E2 -13677.686} C_VEL
LIN {X 0,Y 348.13,Z 312.112,A -85,B 0,C 180,E1 -13681.157,E2 -13681.157} C_VEL
LIN {X 0,Y 348.171,Z 312.104,A -85,B 0,C 180,E1 -13682.314,E2 -13682.314} C_VEL
LIN {X 0,Y 348.059,Z 312.117,A -85,B 0,C 180,E1 -13686.959,E2 -13686.959} C_VEL
LIN {X 0,Y 347.885,Z 312.149,A -85,B 0,C 180,E1 -13690.476,E2 -13690.476} C_VEL
LIN {X 0,Y 347.891,Z 312.138,A -85,B 0,C 180,E1 -13694.15,E2 -13694.15} C_VEL
LIN {X 0,Y 347.822,Z 312.144,A -85,B 0,C 180,E1 -13698.26,E2 -13698.26} C_VEL
LIN {X 0,Y 347.759,Z 312.16,A -85,B 0,C 180,E1 -13701.627,E2 -13701.627} C_VEL
LIN {X 0,Y 347.732,Z 312.169,A -85,B 0,C 180,E1 -13705.115,E2 -13705.115} C_VEL
LIN {X 0,Y 347.73,Z 312.162,A -85,B 0,C 180,E1 -13707.701,E2 -13707.701} C_VEL
LIN {X 0,Y 347.734,Z 312.167,A -85,B 0,C 180,E1 -13710.35,E2 -13710.35} C_VEL
LIN {X 0,Y 347.742,Z 312.167,A -85,B 0,C 180,E1 -13714.045,E2 -13714.045} C_VEL
LIN {X 0,Y 347.751,Z 312.169,A -85,B 0,C 180,E1 -13717.323,E2 -13717.323} C_VEL
LIN {X 0,Y 347.736,Z 312.165,A -85,B 0,C 180,E1 -13721.602,E2 -13721.602} C_VEL
LIN {X 0,Y 347.701,Z 312.171,A -85,B 0,C 180,E1 -13725.028,E2 -13725.028} C_VEL
LIN {X 0,Y 347.746,Z 312.173,A -85,B 0,C 180,E1 -13728.399,E2 -13728.399} C_VEL
LIN {X 0,Y 347.769,Z 312.168,A -85,B 0,C 180,E1 -13732.013,E2 -13732.013} C_VEL
LIN {X 0,Y 347.742,Z 312.162,A -85,B 0,C 180,E1 -13735.537,E2 -13735.537} C_VEL
LIN {X 0,Y 347.768,Z 312.279,A -85,B 0,C 180,E1 -13737.965,E2 -13737.965} C_VEL
LIN {X 0,Y 350.483,Z 323.35,A -85,B 0,C 180,E1 -13741.234,E2 -13741.234} C_VEL
LIN {X 0,Y 352.465,Z 333.238,A -85,B 0,C 180,E1 -13743.982,E2 -13743.982} C_VEL
LIN {X 0,Y 352.784,Z 336.966,A -85,B 0,C 180,E1 -13744.956,E2 -13744.956} C_VEL
LIN {X 0,Y 352.273,Z 340.701,A -85,B 0,C 180,E1 -13745.855,E2 -13745.855} C_VEL
LIN {X 0,Y 357.483,Z 365.28,A -85,B 0,C 180,E1 -13746.848,E2 -13746.848} C_VEL
LIN {X 0,Y 359.424,Z 377.971,A -85,B 0,C 180,E1 -13747.285,E2 -13747.285} C_VEL
LIN {X 0,Y 357.841,Z 449.491,A -85,B 0,C 180,E1 -13748.771,E2 -13748.771} C_VEL
LIN {X 0,Y 356.981,Z 462.524,A -85,B 0,C 180,E1 -13749.246,E2 -13749.246} C_VEL
LIN {X 0,Y 355.983,Z 475.089,A -85,B 0,C 180,E1 -13749.94,E2 -13749.94} C_VEL
LIN {X 0,Y 354.798,Z 486.314,A -85,B 0,C 180,E1 -13750.774,E2 -13750.774} C_VEL
LIN {X 0,Y 353.361,Z 497.92,A -85,B 0,C 180,E1 -13751.896,E2 -13751.896} C_VEL
LIN {X 0,Y 351.838,Z 508.383,A -85,B 0,C 180,E1 -13753.165,E2 -13753.165} C_VEL
LIN {X 0,Y 350.762,Z 515.969,A -85,B 0,C 180,E1 -13754.292,E2 -13754.292} C_VEL
LIN {X 0,Y 349.648,Z 524.118,A -85,B 0,C 180,E1 -13755.747,E2 -13755.747} C_VEL
LIN {X 0,Y 348.371,Z 532.055,A -85,B 0,C 180,E1 -13757.476,E2 -13757.476} C_VEL
LIN {X 0,Y 347.665,Z 537.439,A -85,B 0,C 180,E1 -13758.929,E2 -13758.929} C_VEL
LIN {X 0,Y 346.954,Z 542.731,A -85,B 0,C 180,E1 -13760.675,E2 -13760.675} C_VEL
LIN {X 0,Y 346.495,Z 546.868,A -85,B 0,C 180,E1 -13762.425,E2 -13762.425} C_VEL
LIN {X 0,Y 346.25,Z 549.966,A -85,B 0,C 180,E1 -13764.176,E2 -13764.176} C_VEL
LIN {X 0,Y 346.164,Z 551.518,A -85,B 0,C 180,E1 -13765.343,E2 -13765.343} C_VEL
LIN {X 0,Y 346.141,Z 552.627,A -85,B 0,C 180,E1 -13766.509,E2 -13766.509} C_VEL
LIN {X 0,Y 346.103,Z 553.656,A -85,B 0,C 180,E1 -13768.838,E2 -13768.838} C_VEL
LIN {X 0,Y 346.165,Z 553.596,A -85,B 0,C 180,E1 -13770.001,E2 -13770.001} C_VEL
LIN {X 0,Y 346.123,Z 553.111,A -85,B 0,C 180,E1 -13771.165,E2 -13771.165} C_VEL
LIN {X 0,Y 346.149,Z 550.913,A -85,B 0,C 180,E1 -13773.493,E2 -13773.493} C_VEL
LIN {X 0,Y 346.194,Z 547.68,A -85,B 0,C 180,E1 -13775.497,E2 -13775.497} C_VEL
LIN {X 0,Y 346.438,Z 542.838,A -85,B 0,C 180,E1 -13777.578,E2 -13777.578} C_VEL
LIN {X 0,Y 346.846,Z 536.45,A -85,B 0,C 180,E1 -13779.624,E2 -13779.624} C_VEL
LIN {X 0,Y 347.42,Z 529.48,A -85,B 0,C 180,E1 -13781.376,E2 -13781.376} C_VEL
LIN {X 0,Y 348.355,Z 520.737,A -85,B 0,C 180,E1 -13783.12,E2 -13783.12} C_VEL
LIN {X 0,Y 349.27,Z 511.8,A -85,B 0,C 180,E1 -13784.562,E2 -13784.562} C_VEL
LIN {X 0,Y 350.011,Z 502.209,A -85,B 0,C 180,E1 -13785.834,E2 -13785.834} C_VEL
LIN {X 0,Y 351.116,Z 490.971,A -85,B 0,C 180,E1 -13787.023,E2 -13787.023} C_VEL
LIN {X 0,Y 352.13,Z 478.725,A -85,B 0,C 180,E1 -13788.021,E2 -13788.021} C_VEL
LIN {X 0,Y 352.984,Z 465.893,A -85,B 0,C 180,E1 -13788.803,E2 -13788.803} C_VEL
LIN {X 0,Y 353.681,Z 453.098,A -85,B 0,C 180,E1 -13789.329,E2 -13789.329} C_VEL
LIN {X 0,Y 354.099,Z 435.512,A -85,B 0,C 180,E1 -13789.746,E2 -13789.746} C_VEL
LIN {X 0,Y 354.924,Z 375.109,A -85,B 0,C 180,E1 -13790.97,E2 -13790.97} C_VEL
LIN {X 0,Y 350.048,Z 341.249,A -85,B 0,C 180,E1 -13791.947,E2 -13791.947} C_VEL
LIN {X 0,Y 351.066,Z 330.235,A -85,B 0,C 180,E1 -13794.545,E2 -13794.545} C_VEL
LIN {X 0,Y 349.348,Z 319.646,A -85,B 0,C 180,E1 -13797.238,E2 -13797.238} C_VEL
LIN {X 0,Y 347.807,Z 312.159,A -85,B 0,C 180,E1 -13799.236,E2 -13799.236} C_VEL
LIN {X 0,Y 347.737,Z 312.165,A -85,B 0,C 180,E1 -13803.073,E2 -13803.073} C_VEL
LIN {X 0,Y 347.774,Z 312.167,A -85,B 0,C 180,E1 -13806.065,E2 -13806.065} C_VEL
LIN {X 0,Y 347.735,Z 312.166,A -85,B 0,C 180,E1 -13808.796,E2 -13808.796} C_VEL
LIN {X 0,Y 347.748,Z 312.166,A -85,B 0,C 180,E1 -13811.832,E2 -13811.832} C_VEL
LIN {X 0,Y 347.71,Z 312.169,A -85,B 0,C 180,E1 -13815.027,E2 -13815.027} C_VEL
LIN {X 0,Y 347.751,Z 312.169,A -85,B 0,C 180,E1 -13818.398,E2 -13818.398} C_VEL
LIN {X 0,Y 347.776,Z 312.161,A -85,B 0,C 180,E1 -13822.012,E2 -13822.012} C_VEL
LIN {X 0,Y 347.749,Z 312.164,A -85,B 0,C 180,E1 -13825.536,E2 -13825.536} C_VEL
LIN {X 0,Y 347.749,Z 312.165,A -85,B 0,C 180,E1 -13828.301,E2 -13828.301} C_VEL
LIN {X 0,Y 347.762,Z 312.169,A -85,B 0,C 180,E1 -13830.986,E2 -13830.986} C_VEL
LIN {X 0,Y 347.797,Z 312.162,A -85,B 0,C 180,E1 -13834.89,E2 -13834.89} C_VEL
LIN {X 0,Y 347.785,Z 312.16,A -85,B 0,C 180,E1 -13838.669,E2 -13838.669} C_VEL
LIN {X 0,Y 347.848,Z 312.151,A -85,B 0,C 180,E1 -13842.358,E2 -13842.358} C_VEL
LIN {X 0,Y 347.902,Z 312.147,A -85,B 0,C 180,E1 -13845.971,E2 -13845.971} C_VEL
LIN {X 0,Y 347.931,Z 312.146,A -85,B 0,C 180,E1 -13849.525,E2 -13849.525} C_VEL
LIN {X 0,Y 348.08,Z 312.123,A -85,B 0,C 180,E1 -13853.042,E2 -13853.042} C_VEL
LIN {X 0,Y 348.198,Z 312.111,A -85,B 0,C 180,E1 -13857.686,E2 -13857.686} C_VEL
LIN {X 0,Y 348.306,Z 312.1,A -85,B 0,C 180,E1 -13860,E2 -13860} C_VEL
LIN {X 0,Y 348.2,Z 312.113,A -85,B 0,C 180,E1 -13862.313,E2 -13862.313} C_VEL
LIN {X 0,Y 348.059,Z 312.126,A -85,B 0,C 180,E1 -13866.958,E2 -13866.958} C_VEL
LIN {X 0,Y 347.9,Z 312.152,A -85,B 0,C 180,E1 -13870.475,E2 -13870.475} C_VEL
LIN {X 0,Y 347.902,Z 312.146,A -85,B 0,C 180,E1 -13874.149,E2 -13874.149} C_VEL
LIN {X 0,Y 347.832,Z 312.155,A -85,B 0,C 180,E1 -13878.259,E2 -13878.259} C_VEL
LIN {X 0,Y 347.771,Z 312.162,A -85,B 0,C 180,E1 -13881.626,E2 -13881.626} C_VEL
LIN {X 0,Y 347.796,Z 312.164,A -85,B 0,C 180,E1 -13885.109,E2 -13885.109} C_VEL
LIN {X 0,Y 347.76,Z 312.167,A -85,B 0,C 180,E1 -13889.014,E2 -13889.014} C_VEL
LIN {X 0,Y 347.736,Z 312.169,A -85,B 0,C 180,E1 -13893.072,E2 -13893.072} C_VEL
LIN {X 0,Y 347.773,Z 312.162,A -85,B 0,C 180,E1 -13896.064,E2 -13896.064} C_VEL
LIN {X 0,Y 347.755,Z 312.163,A -85,B 0,C 180,E1 -13898.792,E2 -13898.792} C_VEL
LIN {X 0,Y 347.75,Z 312.169,A -85,B 0,C 180,E1 -13901.83,E2 -13901.83} C_VEL
LIN {X 0,Y 347.707,Z 312.169,A -85,B 0,C 180,E1 -13905.026,E2 -13905.026} C_VEL
LIN {X 0,Y 347.749,Z 312.166,A -85,B 0,C 180,E1 -13908.397,E2 -13908.397} C_VEL
LIN {X 0,Y 347.766,Z 312.168,A -85,B 0,C 180,E1 -13912.013,E2 -13912.013} C_VEL
LIN {X 0,Y 347.746,Z 312.165,A -85,B 0,C 180,E1 -13915.535,E2 -13915.535} C_VEL
LIN {X 0,Y 347.747,Z 312.171,A -85,B 0,C 180,E1 -13918.3,E2 -13918.3} C_VEL
LIN {X 0,Y 347.758,Z 312.164,A -85,B 0,C 180,E1 -13920.985,E2 -13920.985} C_VEL
LIN {X 0,Y 347.795,Z 312.162,A -85,B 0,C 180,E1 -13924.889,E2 -13924.889} C_VEL
LIN {X 0,Y 347.822,Z 312.161,A -85,B 0,C 180,E1 -13928.671,E2 -13928.671} C_VEL
LIN {X 0,Y 347.844,Z 312.154,A -85,B 0,C 180,E1 -13932.357,E2 -13932.357} C_VEL
LIN {X 0,Y 347.898,Z 312.145,A -85,B 0,C 180,E1 -13935.97,E2 -13935.97} C_VEL
LIN {X 0,Y 347.9,Z 312.151,A -85,B 0,C 180,E1 -13939.082,E2 -13939.082} C_VEL
LIN {X 0,Y 349.956,Z 322.968,A -85,B 0,C 180,E1 -13942.071,E2 -13942.071} C_VEL
LIN {X 0,Y 350.115,Z 323.79,A -85,B 0,C 180,E1 -13942.151,E2 -13942.151} C_VEL
LIN {X 0,Y 354.11,Z 343.292,A -85,B 0,C 180,E1 -13942.775,E2 -13942.775} C_VEL
LIN {X 0,Y 355.309,Z 350.129,A -85,B 0,C 180,E1 -13942.981,E2 -13942.981} C_VEL
LIN {X 0,Y 353.914,Z 430.444,A -85,B 0,C 180,E1 -13944.622,E2 -13944.622} C_VEL
LIN {X 0,Y 353.437,Z 442.898,A -85,B 0,C 180,E1 -13945.08,E2 -13945.08} C_VEL
LIN {X 0,Y 352.749,Z 456.297,A -85,B 0,C 180,E1 -13945.82,E2 -13945.82} C_VEL
LIN {X 0,Y 351.945,Z 467.874,A -85,B 0,C 180,E1 -13946.693,E2 -13946.693} C_VEL
LIN {X 0,Y 350.952,Z 479.612,A -85,B 0,C 180,E1 -13947.847,E2 -13947.847} C_VEL
LIN {X 0,Y 349.955,Z 490.041,A -85,B 0,C 180,E1 -13949.136,E2 -13949.136} C_VEL
LIN {X 0,Y 348.959,Z 499.437,A -85,B 0,C 180,E1 -13950.576,E2 -13950.576} C_VEL
LIN {X 0,Y 347.997,Z 508.501,A -85,B 0,C 180,E1 -13952.314,E2 -13952.314} C_VEL
LIN {X 0,Y 347.313,Z 515.8,A -85,B 0,C 180,E1 -13954.06,E2 -13954.06} C_VEL
LIN {X 0,Y 346.898,Z 521.638,A -85,B 0,C 180,E1 -13955.813,E2 -13955.813} C_VEL
LIN {X 0,Y 346.521,Z 526.247,A -85,B 0,C 180,E1 -13957.574,E2 -13957.574} C_VEL
LIN {X 0,Y 346.226,Z 529.759,A -85,B 0,C 180,E1 -13959.345,E2 -13959.345} C_VEL
LIN {X 0,Y 346.097,Z 531.509,A -85,B 0,C 180,E1 -13960.529,E2 -13960.529} C_VEL
LIN {X 0,Y 346.058,Z 532.841,A -85,B 0,C 180,E1 -13961.716,E2 -13961.716} C_VEL
LIN {X 0,Y 346.049,Z 533.772,A -85,B 0,C 180,E1 -13962.908,E2 -13962.908} C_VEL
LIN {X 0,Y 346.007,Z 534.274,A -85,B 0,C 180,E1 -13964.106,E2 -13964.106} C_VEL
LIN {X 0,Y 345.969,Z 534.344,A -85,B 0,C 180,E1 -13965.311,E2 -13965.311} C_VEL
LIN {X 0,Y 346.159,Z 533.49,A -85,B 0,C 180,E1 -13967.402,E2 -13967.402} C_VEL
LIN {X 0,Y 346.339,Z 532.045,A -85,B 0,C 180,E1 -13968.945,E2 -13968.945} C_VEL
LIN {X 0,Y 346.872,Z 528.532,A -85,B 0,C 180,E1 -13971.25,E2 -13971.25} C_VEL
LIN {X 0,Y 347.514,Z 524.13,A -85,B 0,C 180,E1 -13973.225,E2 -13973.225} C_VEL
LIN {X 0,Y 348.357,Z 518.677,A -85,B 0,C 180,E1 -13975.065,E2 -13975.065} C_VEL
LIN {X 0,Y 349.412,Z 511.74,A -85,B 0,C 180,E1 -13976.907,E2 -13976.907} C_VEL
LIN {X 0,Y 350.589,Z 504.293,A -85,B 0,C 180,E1 -13978.493,E2 -13978.493} C_VEL
LIN {X 0,Y 351.767,Z 495.878,A -85,B 0,C 180,E1 -13979.964,E2 -13979.964} C_VEL
LIN {X 0,Y 353.175,Z 486.253,A -85,B 0,C 180,E1 -13981.322,E2 -13981.322} C_VEL
LIN {X 0,Y 354.531,Z 475.614,A -85,B 0,C 180,E1 -13982.526,E2 -13982.526} C_VEL
LIN {X 0,Y 355.379,Z 468.411,A -85,B 0,C 180,E1 -13983.2,E2 -13983.2} C_VEL
LIN {X 0,Y 355.349,Z 463.269,A -85,B 0,C 180,E1 -13983.673,E2 -13983.673} C_VEL
LIN {X 0,Y 353.508,Z 454.835,A -85,B 0,C 180,E1 -13984.467,E2 -13984.467} C_VEL
LIN {X 0,Y 351.5,Z 446.101,A -85,B 0,C 180,E1 -13985.153,E2 -13985.153} C_VEL
LIN {X 0,Y 351.191,Z 440.495,A -85,B 0,C 180,E1 -13985.447,E2 -13985.447} C_VEL
LIN {X 0,Y 351.83,Z 426.769,A -85,B 0,C 180,E1 -13985.883,E2 -13985.883} C_VEL
LIN {X 0,Y 353.594,Z 353.482,A -85,B 0,C 180,E1 -13987.4,E2 -13987.4} C_VEL
LIN {X 0,Y 350.808,Z 341.012,A -85,B 0,C 180,E1 -13987.924,E2 -13987.924} C_VEL
LIN {X 0,Y 343.237,Z 323.629,A -85,B 0,C 180,E1 -13989.026,E2 -13989.026} C_VEL
LIN {X 0,Y 340.683,Z 313.047,A -85,B 0,C 180,E1 -13992.332,E2 -13992.332} C_VEL
LIN {X 0,Y 340.644,Z 313.051,A -85,B 0,C 180,E1 -13996.226,E2 -13996.226} C_VEL
LIN {X 0,Y 340.664,Z 313.05,A -85,B 0,C 180,E1 -13998.687,E2 -13998.687} C_VEL
LIN {X 0,Y 340.711,Z 313.043,A -85,B 0,C 180,E1 -14001.77,E2 -14001.77} C_VEL
LIN {X 0,Y 340.715,Z 313.025,A -85,B 0,C 180,E1 -14005.595,E2 -14005.595} C_VEL
LIN {X 0,Y 340.685,Z 313.048,A -85,B 0,C 180,E1 -14008.954,E2 -14008.954} C_VEL
LIN {X 0,Y 340.711,Z 313.044,A -85,B 0,C 180,E1 -14013.012,E2 -14013.012} C_VEL
LIN {X 0,Y 340.697,Z 313.044,A -85,B 0,C 180,E1 -14016.925,E2 -14016.925} C_VEL
LIN {X 0,Y 340.699,Z 313.043,A -85,B 0,C 180,E1 -14020.728,E2 -14020.728} C_VEL
LIN {X 0,Y 340.783,Z 313.034,A -85,B 0,C 180,E1 -14024.449,E2 -14024.449} C_VEL
LIN {X 0,Y 340.835,Z 313.025,A -85,B 0,C 180,E1 -14028.101,E2 -14028.101} C_VEL
LIN {X 0,Y 340.971,Z 312.999,A -85,B 0,C 180,E1 -14031.705,E2 -14031.705} C_VEL
LIN {X 0,Y 340.999,Z 313.009,A -85,B 0,C 180,E1 -14034.085,E2 -14034.085} C_VEL
LIN {X 0,Y 341.086,Z 312.987,A -85,B 0,C 180,E1 -14037.638,E2 -14037.638} C_VEL
LIN {X 0,Y 341.099,Z 312.987,A -85,B 0,C 180,E1 -14041.181,E2 -14041.181} C_VEL
LIN {X 0,Y 341.107,Z 312.983,A -85,B 0,C 180,E1 -14042.362,E2 -14042.362} C_VEL
LIN {X 0,Y 341.014,Z 313.004,A -85,B 0,C 180,E1 -14045.915,E2 -14045.915} C_VEL
LIN {X 0,Y 340.955,Z 313,A -85,B 0,C 180,E1 -14048.357,E2 -14048.357} C_VEL
LIN {X 0,Y 340.839,Z 313.021,A -85,B 0,C 180,E1 -14051.9,E2 -14051.9} C_VEL
LIN {X 0,Y 340.809,Z 313.028,A -85,B 0,C 180,E1 -14055.55,E2 -14055.55} C_VEL
LIN {X 0,Y 340.755,Z 313.031,A -85,B 0,C 180,E1 -14059.269,E2 -14059.269} C_VEL
LIN {X 0,Y 340.698,Z 313.036,A -85,B 0,C 180,E1 -14063.075,E2 -14063.075} C_VEL
LIN {X 0,Y 340.712,Z 313.038,A -85,B 0,C 180,E1 -14066.988,E2 -14066.988} C_VEL
LIN {X 0,Y 340.688,Z 313.044,A -85,B 0,C 180,E1 -14071.046,E2 -14071.046} C_VEL
LIN {X 0,Y 340.712,Z 313.04,A -85,B 0,C 180,E1 -14075.28,E2 -14075.28} C_VEL
LIN {X 0,Y 340.688,Z 313.042,A -85,B 0,C 180,E1 -14078.384,E2 -14078.384} C_VEL
LIN {X 0,Y 340.688,Z 313.038,A -85,B 0,C 180,E1 -14082.046,E2 -14082.046} C_VEL
LIN {X 0,Y 340.648,Z 313.057,A -85,B 0,C 180,E1 -14086.228,E2 -14086.228} C_VEL
LIN {X 0,Y 340.683,Z 313.05,A -85,B 0,C 180,E1 -14089.755,E2 -14089.755} C_VEL
LIN {X 0,Y 340.701,Z 313.045,A -85,B 0,C 180,E1 -14093.26,E2 -14093.26} C_VEL
LIN {X 0,Y 340.7,Z 313.048,A -85,B 0,C 180,E1 -14096.864,E2 -14096.864} C_VEL
LIN {X 0,Y 340.728,Z 313.126,A -85,B 0,C 180,E1 -14097.395,E2 -14097.395} C_VEL
LIN {X 0,Y 343.321,Z 323.549,A -85,B 0,C 180,E1 -14100.576,E2 -14100.576} C_VEL
LIN {X 0,Y 345.459,Z 333.855,A -85,B 0,C 180,E1 -14103.526,E2 -14103.526} C_VEL
LIN {X 0,Y 345.943,Z 338.387,A -85,B 0,C 180,E1 -14104.748,E2 -14104.748} C_VEL
LIN {X 0,Y 345.686,Z 340.492,A -85,B 0,C 180,E1 -14105.268,E2 -14105.268} C_VEL
LIN {X 0,Y 351.207,Z 366.704,A -85,B 0,C 180,E1 -14106.36,E2 -14106.36} C_VEL
LIN {X 0,Y 353.082,Z 378.371,A -85,B 0,C 180,E1 -14106.781,E2 -14106.781} C_VEL
LIN {X 0,Y 351.415,Z 449.537,A -85,B 0,C 180,E1 -14108.287,E2 -14108.287} C_VEL
LIN {X 0,Y 350.531,Z 462.486,A -85,B 0,C 180,E1 -14108.769,E2 -14108.769} C_VEL
LIN {X 0,Y 349.485,Z 475.01,A -85,B 0,C 180,E1 -14109.474,E2 -14109.474} C_VEL
LIN {X 0,Y 348.138,Z 486.991,A -85,B 0,C 180,E1 -14110.391,E2 -14110.391} C_VEL
LIN {X 0,Y 346.657,Z 498.429,A -85,B 0,C 180,E1 -14111.533,E2 -14111.533} C_VEL
LIN {X 0,Y 345.063,Z 508.763,A -85,B 0,C 180,E1 -14112.824,E2 -14112.824} C_VEL
LIN {X 0,Y 343.867,Z 516.739,A -85,B 0,C 180,E1 -14114.054,E2 -14114.054} C_VEL
LIN {X 0,Y 342.547,Z 525.75,A -85,B 0,C 180,E1 -14115.748,E2 -14115.748} C_VEL
LIN {X 0,Y 341.271,Z 533.282,A -85,B 0,C 180,E1 -14117.513,E2 -14117.513} C_VEL
LIN {X 0,Y 340.384,Z 539.364,A -85,B 0,C 180,E1 -14119.292,E2 -14119.292} C_VEL
LIN {X 0,Y 339.756,Z 544.205,A -85,B 0,C 180,E1 -14121.076,E2 -14121.076} C_VEL
LIN {X 0,Y 339.323,Z 547.942,A -85,B 0,C 180,E1 -14122.862,E2 -14122.862} C_VEL
LIN {X 0,Y 339.17,Z 549.881,A -85,B 0,C 180,E1 -14124.054,E2 -14124.054} C_VEL
LIN {X 0,Y 339.07,Z 551.402,A -85,B 0,C 180,E1 -14125.245,E2 -14125.245} C_VEL
LIN {X 0,Y 339.065,Z 552.479,A -85,B 0,C 180,E1 -14126.436,E2 -14126.436} C_VEL
LIN {X 0,Y 339.006,Z 553.467,A -85,B 0,C 180,E1 -14128.813,E2 -14128.813} C_VEL
LIN {X 0,Y 339.068,Z 553.383,A -85,B 0,C 180,E1 -14130.001,E2 -14130.001} C_VEL
LIN {X 0,Y 339.025,Z 552.86,A -85,B 0,C 180,E1 -14131.189,E2 -14131.189} C_VEL
LIN {X 0,Y 339.075,Z 550.621,A -85,B 0,C 180,E1 -14133.566,E2 -14133.566} C_VEL
LIN {X 0,Y 339.093,Z 547.678,A -85,B 0,C 180,E1 -14135.426,E2 -14135.426} C_VEL
LIN {X 0,Y 339.27,Z 543.959,A -85,B 0,C 180,E1 -14137.141,E2 -14137.141} C_VEL
LIN {X 0,Y 339.589,Z 538.961,A -85,B 0,C 180,E1 -14138.93,E2 -14138.93} C_VEL
LIN {X 0,Y 340.094,Z 532.664,A -85,B 0,C 180,E1 -14140.719,E2 -14140.719} C_VEL
LIN {X 0,Y 340.862,Z 524.769,A -85,B 0,C 180,E1 -14142.504,E2 -14142.504} C_VEL
LIN {X 0,Y 341.701,Z 516.699,A -85,B 0,C 180,E1 -14143.986,E2 -14143.986} C_VEL
LIN {X 0,Y 342.682,Z 506.834,A -85,B 0,C 180,E1 -14145.464,E2 -14145.464} C_VEL
LIN {X 0,Y 343.683,Z 495.817,A -85,B 0,C 180,E1 -14146.79,E2 -14146.79} C_VEL
LIN {X 0,Y 344.738,Z 485.023,A -85,B 0,C 180,E1 -14147.807,E2 -14147.807} C_VEL
LIN {X 0,Y 345.693,Z 471.984,A -85,B 0,C 180,E1 -14148.753,E2 -14148.753} C_VEL
LIN {X 0,Y 346.531,Z 459.522,A -85,B 0,C 180,E1 -14149.397,E2 -14149.397} C_VEL
LIN {X 0,Y 347.019,Z 446.534,A -85,B 0,C 180,E1 -14149.831,E2 -14149.831} C_VEL
LIN {X 0,Y 348.179,Z 376.041,A -85,B 0,C 180,E1 -14151.292,E2 -14151.292} C_VEL
LIN {X 0,Y 343.18,Z 340.948,A -85,B 0,C 180,E1 -14152.346,E2 -14152.346} C_VEL
LIN {X 0,Y 344.07,Z 330.961,A -85,B 0,C 180,E1 -14154.756,E2 -14154.756} C_VEL
LIN {X 0,Y 341.978,Z 318.895,A -85,B 0,C 180,E1 -14157.908,E2 -14157.908} C_VEL
LIN {X 0,Y 340.741,Z 313.042,A -85,B 0,C 180,E1 -14159.502,E2 -14159.502} C_VEL
LIN {X 0,Y 340.691,Z 313.044,A -85,B 0,C 180,E1 -14162.436,E2 -14162.436} C_VEL
LIN {X 0,Y 340.722,Z 313.04,A -85,B 0,C 180,E1 -14165.279,E2 -14165.279} C_VEL
LIN {X 0,Y 340.698,Z 313.046,A -85,B 0,C 180,E1 -14168.383,E2 -14168.383} C_VEL
LIN {X 0,Y 340.698,Z 313.046,A -85,B 0,C 180,E1 -14172.045,E2 -14172.045} C_VEL
LIN {X 0,Y 340.656,Z 313.052,A -85,B 0,C 180,E1 -14176.227,E2 -14176.227} C_VEL
LIN {X 0,Y 340.689,Z 313.044,A -85,B 0,C 180,E1 -14179.754,E2 -14179.754} C_VEL
LIN {X 0,Y 340.709,Z 313.042,A -85,B 0,C 180,E1 -14183.259,E2 -14183.259} C_VEL
LIN {X 0,Y 340.697,Z 313.043,A -85,B 0,C 180,E1 -14186.154,E2 -14186.154} C_VEL
LIN {X 0,Y 340.736,Z 313.038,A -85,B 0,C 180,E1 -14190.328,E2 -14190.328} C_VEL
LIN {X 0,Y 340.749,Z 313.036,A -85,B 0,C 180,E1 -14194.333,E2 -14194.333} C_VEL
LIN {X 0,Y 340.746,Z 313.036,A -85,B 0,C 180,E1 -14198.207,E2 -14198.207} C_VEL
LIN {X 0,Y 340.797,Z 313.031,A -85,B 0,C 180,E1 -14201.981,E2 -14201.981} C_VEL
LIN {X 0,Y 340.874,Z 313.025,A -85,B 0,C 180,E1 -14205.705,E2 -14205.705} C_VEL
LIN {X 0,Y 340.874,Z 313.022,A -85,B 0,C 180,E1 -14209.306,E2 -14209.306} C_VEL
LIN {X 0,Y 341.048,Z 312.998,A -85,B 0,C 180,E1 -14212.897,E2 -14212.897} C_VEL
LIN {X 0,Y 341.135,Z 312.99,A -85,B 0,C 180,E1 -14217.638,E2 -14217.638} C_VEL
LIN {X 0,Y 341.258,Z 312.978,A -85,B 0,C 180,E1 -14220,E2 -14220} C_VEL
LIN {X 0,Y 341.161,Z 312.989,A -85,B 0,C 180,E1 -14222.361,E2 -14222.361} C_VEL
LIN {X 0,Y 341.006,Z 313.004,A -85,B 0,C 180,E1 -14227.103,E2 -14227.103} C_VEL
LIN {X 0,Y 340.852,Z 313.028,A -85,B 0,C 180,E1 -14230.694,E2 -14230.694} C_VEL
LIN {X 0,Y 340.867,Z 313.024,A -85,B 0,C 180,E1 -14234.324,E2 -14234.324} C_VEL
LIN {X 0,Y 340.789,Z 313.033,A -85,B 0,C 180,E1 -14238.44,E2 -14238.44} C_VEL
LIN {X 0,Y 340.721,Z 313.039,A -85,B 0,C 180,E1 -14241.841,E2 -14241.841} C_VEL
LIN {X 0,Y 340.748,Z 313.037,A -85,B 0,C 180,E1 -14245.666,E2 -14245.666} C_VEL
LIN {X 0,Y 340.735,Z 313.04,A -85,B 0,C 180,E1 -14249.671,E2 -14249.671} C_VEL
LIN {X 0,Y 340.695,Z 313.045,A -85,B 0,C 180,E1 -14253.846,E2 -14253.846} C_VEL
LIN {X 0,Y 340.708,Z 313.041,A -85,B 0,C 180,E1 -14256.741,E2 -14256.741} C_VEL
LIN {X 0,Y 340.687,Z 313.044,A -85,B 0,C 180,E1 -14260.246,E2 -14260.246} C_VEL
LIN {X 0,Y 340.654,Z 313.054,A -85,B 0,C 180,E1 -14263.772,E2 -14263.772} C_VEL
LIN {X 0,Y 340.698,Z 313.048,A -85,B 0,C 180,E1 -14267.954,E2 -14267.954} C_VEL
LIN {X 0,Y 340.722,Z 313.042,A -85,B 0,C 180,E1 -14271.77,E2 -14271.77} C_VEL
LIN {X 0,Y 340.725,Z 313.039,A -85,B 0,C 180,E1 -14275.595,E2 -14275.595} C_VEL
LIN {X 0,Y 340.697,Z 313.043,A -85,B 0,C 180,E1 -14278.954,E2 -14278.954} C_VEL
LIN {X 0,Y 340.712,Z 313.047,A -85,B 0,C 180,E1 -14282.495,E2 -14282.495} C_VEL
LIN {X 0,Y 340.754,Z 313.035,A -85,B 0,C 180,E1 -14285.637,E2 -14285.637} C_VEL
LIN {X 0,Y 340.753,Z 313.036,A -85,B 0,C 180,E1 -14289.474,E2 -14289.474} C_VEL
LIN {X 0,Y 340.793,Z 313.03,A -85,B 0,C 180,E1 -14291.98,E2 -14291.98} C_VEL
LIN {X 0,Y 340.87,Z 313.022,A -85,B 0,C 180,E1 -14295.704,E2 -14295.704} C_VEL
LIN {X 0,Y 340.868,Z 313.159,A -85,B 0,C 180,E1 -14298.854,E2 -14298.854} C_VEL
LIN {X 0,Y 342.824,Z 323.285,A -85,B 0,C 180,E1 -14301.711,E2 -14301.711} C_VEL
LIN {X 0,Y 344.459,Z 329.538,A -85,B 0,C 180,E1 -14301.966,E2 -14301.966} C_VEL
LIN {X 0,Y 348.537,Z 351.077,A -85,B 0,C 180,E1 -14302.649,E2 -14302.649} C_VEL
LIN {X 0,Y 347.101,Z 430.414,A -85,B 0,C 180,E1 -14304.298,E2 -14304.298} C_VEL
LIN {X 0,Y 346.61,Z 442.948,A -85,B 0,C 180,E1 -14304.764,E2 -14304.764} C_VEL
LIN {X 0,Y 345.906,Z 456.227,A -85,B 0,C 180,E1 -14305.508,E2 -14305.508} C_VEL
LIN {X 0,Y 345.04,Z 468.252,A -85,B 0,C 180,E1 -14306.431,E2 -14306.431} C_VEL
LIN {X 0,Y 343.978,Z 480.392,A -85,B 0,C 180,E1 -14307.657,E2 -14307.657} C_VEL
LIN {X 0,Y 342.953,Z 490.72,A -85,B 0,C 180,E1 -14308.972,E2 -14308.972} C_VEL
LIN {X 0,Y 342.01,Z 499.176,A -85,B 0,C 180,E1 -14310.293,E2 -14310.293} C_VEL
LIN {X 0,Y 341.031,Z 508.323,A -85,B 0,C 180,E1 -14312.066,E2 -14312.066} C_VEL
LIN {X 0,Y 340.301,Z 515.69,A -85,B 0,C 180,E1 -14313.847,E2 -14313.847} C_VEL
LIN {X 0,Y 339.873,Z 520.684,A -85,B 0,C 180,E1 -14315.338,E2 -14315.338} C_VEL
LIN {X 0,Y 339.513,Z 525.535,A -85,B 0,C 180,E1 -14317.134,E2 -14317.134} C_VEL
LIN {X 0,Y 339.199,Z 529.272,A -85,B 0,C 180,E1 -14318.939,E2 -14318.939} C_VEL
LIN {X 0,Y 339.003,Z 531.977,A -85,B 0,C 180,E1 -14320.752,E2 -14320.752} C_VEL
LIN {X 0,Y 338.954,Z 533.974,A -85,B 0,C 180,E1 -14322.964,E2 -14322.964} C_VEL
LIN {X 0,Y 338.903,Z 534.506,A -85,B 0,C 180,E1 -14324.408,E2 -14324.408} C_VEL
LIN {X 0,Y 338.881,Z 534.516,A -85,B 0,C 180,E1 -14325.64,E2 -14325.64} C_VEL
LIN {X 0,Y 339.102,Z 533.679,A -85,B 0,C 180,E1 -14327.567,E2 -14327.567} C_VEL
LIN {X 0,Y 339.342,Z 531.973,A -85,B 0,C 180,E1 -14329.351,E2 -14329.351} C_VEL
LIN {X 0,Y 339.885,Z 528.711,A -85,B 0,C 180,E1 -14331.489,E2 -14331.489} C_VEL
LIN {X 0,Y 340.387,Z 525.285,A -85,B 0,C 180,E1 -14333.096,E2 -14333.096} C_VEL
LIN {X 0,Y 341.259,Z 519.998,A -85,B 0,C 180,E1 -14335.022,E2 -14335.022} C_VEL
LIN {X 0,Y 342.29,Z 513.58,A -85,B 0,C 180,E1 -14336.852,E2 -14336.852} C_VEL
LIN {X 0,Y 343.589,Z 505.983,A -85,B 0,C 180,E1 -14338.569,E2 -14338.569} C_VEL
LIN {X 0,Y 344.969,Z 496.613,A -85,B 0,C 180,E1 -14340.279,E2 -14340.279} C_VEL
LIN {X 0,Y 346.475,Z 487.02,A -85,B 0,C 180,E1 -14341.675,E2 -14341.675} C_VEL
LIN {X 0,Y 347.856,Z 476.679,A -85,B 0,C 180,E1 -14342.885,E2 -14342.885} C_VEL
LIN {X 0,Y 349.174,Z 465.141,A -85,B 0,C 180,E1 -14343.953,E2 -14343.953} C_VEL
LIN {X 0,Y 350.312,Z 453.409,A -85,B 0,C 180,E1 -14344.785,E2 -14344.785} C_VEL
LIN {X 0,Y 351.18,Z 440.74,A -85,B 0,C 180,E1 -14345.437,E2 -14345.437} C_VEL
LIN {X 0,Y 351.191,Z 440.495,A -85,B 0,C 180,E1 -14345.447,E2 -14345.447} C_VEL
LIN {X 0,Y 350.921,Z 434.798,A -85,B 0,C 180,E1 -14345.706,E2 -14345.706} C_VEL
LIN {X 0,Y 346.335,Z 416.248,A -85,B 0,C 180,E1 -14346.58,E2 -14346.58} C_VEL
LIN {X 0,Y 345.884,Z 410.448,A -85,B 0,C 180,E1 -14346.747,E2 -14346.747} C_VEL
LIN {X 0,Y 347.278,Z 354.412,A -85,B 0,C 180,E1 -14347.925,E2 -14347.925} C_VEL
LIN {X 0,Y 344.707,Z 343.284,A -85,B 0,C 180,E1 -14348.416,E2 -14348.416} C_VEL
LIN {X 0,Y 337.305,Z 326.725,A -85,B 0,C 180,E1 -14349.512,E2 -14349.512} C_VEL
LIN {X 0,Y 336.044,Z 323.874,A -85,B 0,C 180,E1 -14349.709,E2 -14349.709} C_VEL
LIN {X 0,Y 333.632,Z 313.93,A -85,B 0,C 180,E1 -14352.917,E2 -14352.917} C_VEL
LIN {X 0,Y 333.589,Z 313.932,A -85,B 0,C 180,E1 -14355.954,E2 -14355.954} C_VEL
LIN {X 0,Y 333.595,Z 313.933,A -85,B 0,C 180,E1 -14359.324,E2 -14359.324} C_VEL
LIN {X 0,Y 333.655,Z 313.925,A -85,B 0,C 180,E1 -14363.168,E2 -14363.168} C_VEL
LIN {X 0,Y 333.666,Z 313.905,A -85,B 0,C 180,E1 -14365.341,E2 -14365.341} C_VEL
LIN {X 0,Y 333.621,Z 313.927,A -85,B 0,C 180,E1 -14368.221,E2 -14368.221} C_VEL
LIN {X 0,Y 333.645,Z 313.919,A -85,B 0,C 180,E1 -14371.022,E2 -14371.022} C_VEL
LIN {X 0,Y 333.657,Z 313.919,A -85,B 0,C 180,E1 -14375.085,E2 -14375.085} C_VEL
LIN {X 0,Y 333.645,Z 313.92,A -85,B 0,C 180,E1 -14379.017,E2 -14379.017} C_VEL
LIN {X 0,Y 333.703,Z 313.911,A -85,B 0,C 180,E1 -14381.585,E2 -14381.585} C_VEL
LIN {X 0,Y 333.765,Z 313.905,A -85,B 0,C 180,E1 -14385.6,E2 -14385.6} C_VEL
LIN {X 0,Y 333.804,Z 313.902,A -85,B 0,C 180,E1 -14389.077,E2 -14389.077} C_VEL
LIN {X 0,Y 333.944,Z 313.883,A -85,B 0,C 180,E1 -14392.746,E2 -14392.746} C_VEL
LIN {X 0,Y 333.762,Z 313.904,A -85,B 0,C 180,E1 -14395.169,E2 -14395.169} C_VEL
LIN {X 0,Y 334.029,Z 313.866,A -85,B 0,C 180,E1 -14397.589,E2 -14397.589} C_VEL
LIN {X 0,Y 334.067,Z 313.863,A -85,B 0,C 180,E1 -14401.206,E2 -14401.206} C_VEL
LIN {X 0,Y 334.048,Z 313.862,A -85,B 0,C 180,E1 -14402.412,E2 -14402.412} C_VEL
LIN {X 0,Y 333.988,Z 313.88,A -85,B 0,C 180,E1 -14406.04,E2 -14406.04} C_VEL
LIN {X 0,Y 333.811,Z 313.899,A -85,B 0,C 180,E1 -14409.697,E2 -14409.697} C_VEL
LIN {X 0,Y 333.788,Z 313.893,A -85,B 0,C 180,E1 -14413.392,E2 -14413.392} C_VEL
LIN {X 0,Y 333.711,Z 313.906,A -85,B 0,C 180,E1 -14417.148,E2 -14417.148} C_VEL
LIN {X 0,Y 333.71,Z 313.912,A -85,B 0,C 180,E1 -14419.692,E2 -14419.692} C_VEL
LIN {X 0,Y 333.637,Z 313.917,A -85,B 0,C 180,E1 -14423.593,E2 -14423.593} C_VEL
LIN {X 0,Y 333.661,Z 313.914,A -85,B 0,C 180,E1 -14427.607,E2 -14427.607} C_VEL
LIN {X 0,Y 333.651,Z 313.921,A -85,B 0,C 180,E1 -14430.367,E2 -14430.367} C_VEL
LIN {X 0,Y 333.631,Z 313.925,A -85,B 0,C 180,E1 -14433.209,E2 -14433.209} C_VEL
LIN {X 0,Y 333.669,Z 313.919,A -85,B 0,C 180,E1 -14436.14,E2 -14436.14} C_VEL
LIN {X 0,Y 333.596,Z 313.926,A -85,B 0,C 180,E1 -14439.2,E2 -14439.2} C_VEL
LIN {X 0,Y 333.624,Z 313.913,A -85,B 0,C 180,E1 -14442.5,E2 -14442.5} C_VEL
LIN {X 0,Y 333.592,Z 313.937,A -85,B 0,C 180,E1 -14445.956,E2 -14445.956} C_VEL
LIN {X 0,Y 333.643,Z 313.928,A -85,B 0,C 180,E1 -14449.317,E2 -14449.317} C_VEL
LIN {X 0,Y 333.661,Z 313.923,A -85,B 0,C 180,E1 -14453.169,E2 -14453.169} C_VEL
LIN {X 0,Y 333.663,Z 313.985,A -85,B 0,C 180,E1 -14456.796,E2 -14456.796} C_VEL
LIN {X 0,Y 336.404,Z 325.003,A -85,B 0,C 180,E1 -14460.255,E2 -14460.255} C_VEL
LIN {X 0,Y 338.524,Z 335.073,A -85,B 0,C 180,E1 -14463.217,E2 -14463.217} C_VEL
LIN {X 0,Y 339.077,Z 340.205,A -85,B 0,C 180,E1 -14464.632,E2 -14464.632} C_VEL
LIN {X 0,Y 344.323,Z 364.668,A -85,B 0,C 180,E1 -14465.713,E2 -14465.713} C_VEL
LIN {X 0,Y 346.763,Z 379.176,A -85,B 0,C 180,E1 -14466.266,E2 -14466.266} C_VEL
LIN {X 0,Y 345.025,Z 449.578,A -85,B 0,C 180,E1 -14467.785,E2 -14467.785} C_VEL
LIN {X 0,Y 344.112,Z 462.447,A -85,B 0,C 180,E1 -14468.275,E2 -14468.275} C_VEL
LIN {X 0,Y 343.007,Z 474.931,A -85,B 0,C 180,E1 -14468.989,E2 -14468.989} C_VEL
LIN {X 0,Y 341.737,Z 486.087,A -85,B 0,C 180,E1 -14469.852,E2 -14469.852} C_VEL
LIN {X 0,Y 340.276,Z 496.379,A -85,B 0,C 180,E1 -14470.861,E2 -14470.861} C_VEL
LIN {X 0,Y 338.625,Z 507.027,A -85,B 0,C 180,E1 -14472.175,E2 -14472.175} C_VEL
LIN {X 0,Y 337.217,Z 515.581,A -85,B 0,C 180,E1 -14473.476,E2 -14473.476} C_VEL
LIN {X 0,Y 335.912,Z 524.52,A -85,B 0,C 180,E1 -14475.151,E2 -14475.151} C_VEL
LIN {X 0,Y 334.506,Z 532.277,A -85,B 0,C 180,E1 -14476.948,E2 -14476.948} C_VEL
LIN {X 0,Y 333.405,Z 539.411,A -85,B 0,C 180,E1 -14479.065,E2 -14479.065} C_VEL
LIN {X 0,Y 332.728,Z 544.196,A -85,B 0,C 180,E1 -14480.886,E2 -14480.886} C_VEL
LIN {X 0,Y 332.264,Z 547.882,A -85,B 0,C 180,E1 -14482.71,E2 -14482.71} C_VEL
LIN {X 0,Y 332.066,Z 550.067,A -85,B 0,C 180,E1 -14484.119,E2 -14484.119} C_VEL
LIN {X 0,Y 331.969,Z 552.331,A -85,B 0,C 180,E1 -14486.36,E2 -14486.36} C_VEL
LIN {X 0,Y 331.912,Z 553.279,A -85,B 0,C 180,E1 -14488.788,E2 -14488.788} C_VEL
LIN {X 0,Y 331.971,Z 553.16,A -85,B 0,C 180,E1 -14490.001,E2 -14490.001} C_VEL
LIN {X 0,Y 331.93,Z 552.609,A -85,B 0,C 180,E1 -14491.214,E2 -14491.214} C_VEL
LIN {X 0,Y 332.001,Z 550.328,A -85,B 0,C 180,E1 -14493.642,E2 -14493.642} C_VEL
LIN {X 0,Y 332.084,Z 546.624,A -85,B 0,C 180,E1 -14495.912,E2 -14495.912} C_VEL
LIN {X 0,Y 332.31,Z 542.018,A -85,B 0,C 180,E1 -14497.902,E2 -14497.902} C_VEL
LIN {X 0,Y 332.787,Z 535.525,A -85,B 0,C 180,E1 -14500.035,E2 -14500.035} C_VEL
LIN {X 0,Y 333.422,Z 528.394,A -85,B 0,C 180,E1 -14501.861,E2 -14501.861} C_VEL
LIN {X 0,Y 334.382,Z 519.475,A -85,B 0,C 180,E1 -14503.678,E2 -14503.678} C_VEL
LIN {X 0,Y 335.326,Z 511.321,A -85,B 0,C 180,E1 -14505.032,E2 -14505.032} C_VEL
LIN {X 0,Y 336.194,Z 501.392,A -85,B 0,C 180,E1 -14506.393,E2 -14506.393} C_VEL
LIN {X 0,Y 337.295,Z 490.474,A -85,B 0,C 180,E1 -14507.586,E2 -14507.586} C_VEL
LIN {X 0,Y 338.398,Z 478.2,A -85,B 0,C 180,E1 -14508.622,E2 -14508.622} C_VEL
LIN {X 0,Y 339.332,Z 465.322,A -85,B 0,C 180,E1 -14509.432,E2 -14509.432} C_VEL
LIN {X 0,Y 340.046,Z 452.388,A -85,B 0,C 180,E1 -14509.979,E2 -14509.979} C_VEL
LIN {X 0,Y 340.507,Z 434.07,A -85,B 0,C 180,E1 -14510.424,E2 -14510.424} C_VEL
LIN {X 0,Y 341.313,Z 376.463,A -85,B 0,C 180,E1 -14511.639,E2 -14511.639} C_VEL
LIN {X 0,Y 336.276,Z 340.855,A -85,B 0,C 180,E1 -14512.713,E2 -14512.713} C_VEL
LIN {X 0,Y 337.054,Z 332.986,A -85,B 0,C 180,E1 -14514.648,E2 -14514.648} C_VEL
LIN {X 0,Y 336.378,Z 327.61,A -85,B 0,C 180,E1 -14516.05,E2 -14516.05} C_VEL
LIN {X 0,Y 334.384,Z 317.035,A -85,B 0,C 180,E1 -14518.909,E2 -14518.909} C_VEL
LIN {X 0,Y 333.701,Z 313.921,A -85,B 0,C 180,E1 -14519.821,E2 -14519.821} C_VEL
LIN {X 0,Y 333.641,Z 313.922,A -85,B 0,C 180,E1 -14523.209,E2 -14523.209} C_VEL
LIN {X 0,Y 333.679,Z 313.922,A -85,B 0,C 180,E1 -14526.14,E2 -14526.14} C_VEL
LIN {X 0,Y 333.606,Z 313.926,A -85,B 0,C 180,E1 -14529.199,E2 -14529.199} C_VEL
LIN {X 0,Y 333.633,Z 313.927,A -85,B 0,C 180,E1 -14532.5,E2 -14532.5} C_VEL
LIN {X 0,Y 333.6,Z 313.929,A -85,B 0,C 180,E1 -14535.955,E2 -14535.955} C_VEL
LIN {X 0,Y 333.65,Z 313.921,A -85,B 0,C 180,E1 -14539.316,E2 -14539.316} C_VEL
LIN {X 0,Y 333.669,Z 313.92,A -85,B 0,C 180,E1 -14543.168,E2 -14543.168} C_VEL
LIN {X 0,Y 333.679,Z 313.918,A -85,B 0,C 180,E1 -14545.341,E2 -14545.341} C_VEL
LIN {X 0,Y 333.634,Z 313.923,A -85,B 0,C 180,E1 -14548.222,E2 -14548.222} C_VEL
LIN {X 0,Y 333.675,Z 313.924,A -85,B 0,C 180,E1 -14551.024,E2 -14551.024} C_VEL
LIN {X 0,Y 333.718,Z 313.918,A -85,B 0,C 180,E1 -14555.09,E2 -14555.09} C_VEL
LIN {X 0,Y 333.675,Z 313.92,A -85,B 0,C 180,E1 -14559.019,E2 -14559.019} C_VEL
LIN {X 0,Y 333.745,Z 313.912,A -85,B 0,C 180,E1 -14561.586,E2 -14561.586} C_VEL
LIN {X 0,Y 333.813,Z 313.906,A -85,B 0,C 180,E1 -14565.577,E2 -14565.577} C_VEL
LIN {X 0,Y 333.837,Z 313.897,A -85,B 0,C 180,E1 -14569.078,E2 -14569.078} C_VEL
LIN {X 0,Y 333.995,Z 313.876,A -85,B 0,C 180,E1 -14572.747,E2 -14572.747} C_VEL
LIN {X 0,Y 333.797,Z 313.902,A -85,B 0,C 180,E1 -14575.169,E2 -14575.169} C_VEL
LIN {X 0,Y 334.076,Z 313.869,A -85,B 0,C 180,E1 -14577.588,E2 -14577.588} C_VEL
LIN {X 0,Y 334.21,Z 313.855,A -85,B 0,C 180,E1 -14580,E2 -14580} C_VEL
LIN {X 0,Y 334.098,Z 313.867,A -85,B 0,C 180,E1 -14582.411,E2 -14582.411} C_VEL
LIN {X 0,Y 333.963,Z 313.88,A -85,B 0,C 180,E1 -14586.528,E2 -14586.528} C_VEL
LIN {X 0,Y 333.824,Z 313.899,A -85,B 0,C 180,E1 -14589.696,E2 -14589.696} C_VEL
LIN {X 0,Y 333.8,Z 313.9,A -85,B 0,C 180,E1 -14593.391,E2 -14593.391} C_VEL
LIN {X 0,Y 333.723,Z 313.913,A -85,B 0,C 180,E1 -14597.147,E2 -14597.147} C_VEL
LIN {X 0,Y 333.675,Z 313.917,A -85,B 0,C 180,E1 -14599.694,E2 -14599.694} C_VEL
LIN {X 0,Y 333.671,Z 313.918,A -85,B 0,C 180,E1 -14603.59,E2 -14603.59} C_VEL
LIN {X 0,Y 333.679,Z 313.915,A -85,B 0,C 180,E1 -14606.251,E2 -14606.251} C_VEL
LIN {X 0,Y 333.663,Z 313.918,A -85,B 0,C 180,E1 -14610.365,E2 -14610.365} C_VEL
LIN {X 0,Y 333.64,Z 313.926,A -85,B 0,C 180,E1 -14613.208,E2 -14613.208} C_VEL
LIN {X 0,Y 333.668,Z 313.918,A -85,B 0,C 180,E1 -14616.832,E2 -14616.832} C_VEL
LIN {X 0,Y 333.647,Z 313.92,A -85,B 0,C 180,E1 -14620.767,E2 -14620.767} C_VEL
LIN {X 0,Y 333.595,Z 313.929,A -85,B 0,C 180,E1 -14624.25,E2 -14624.25} C_VEL
LIN {X 0,Y 333.642,Z 313.923,A -85,B 0,C 180,E1 -14627.617,E2 -14627.617} C_VEL
LIN {X 0,Y 333.641,Z 313.921,A -85,B 0,C 180,E1 -14631.204,E2 -14631.204} C_VEL
LIN {X 0,Y 333.677,Z 313.92,A -85,B 0,C 180,E1 -14633.86,E2 -14633.86} C_VEL
LIN {X 0,Y 333.647,Z 313.921,A -85,B 0,C 180,E1 -14637.412,E2 -14637.412} C_VEL
LIN {X 0,Y 333.671,Z 313.919,A -85,B 0,C 180,E1 -14641.023,E2 -14641.023} C_VEL
LIN {X 0,Y 333.715,Z 313.914,A -85,B 0,C 180,E1 -14645.089,E2 -14645.089} C_VEL
LIN {X 0,Y 333.686,Z 313.92,A -85,B 0,C 180,E1 -14649.019,E2 -14649.019} C_VEL
LIN {X 0,Y 333.742,Z 313.909,A -85,B 0,C 180,E1 -14651.586,E2 -14651.586} C_VEL
LIN {X 0,Y 333.809,Z 313.902,A -85,B 0,C 180,E1 -14655.576,E2 -14655.576} C_VEL
LIN {X 0,Y 333.833,Z 314.025,A -85,B 0,C 180,E1 -14658.578,E2 -14658.578} C_VEL
LIN {X 0,Y 335.703,Z 323.585,A -85,B 0,C 180,E1 -14661.332,E2 -14661.332} C_VEL
LIN {X 0,Y 337.965,Z 331.66,A -85,B 0,C 180,E1 -14661.648,E2 -14661.648} C_VEL
LIN {X 0,Y 341.814,Z 352.332,A -85,B 0,C 180,E1 -14662.318,E2 -14662.318} C_VEL
LIN {X 0,Y 340.269,Z 430.979,A -85,B 0,C 180,E1 -14663.984,E2 -14663.984} C_VEL
LIN {X 0,Y 339.745,Z 443.647,A -85,B 0,C 180,E1 -14664.472,E2 -14664.472} C_VEL
LIN {X 0,Y 339.02,Z 456.986,A -85,B 0,C 180,E1 -14665.242,E2 -14665.242} C_VEL
LIN {X 0,Y 338.199,Z 468.029,A -85,B 0,C 180,E1 -14666.109,E2 -14666.109} C_VEL
LIN {X 0,Y 337.135,Z 479.843,A -85,B 0,C 180,E1 -14667.311,E2 -14667.311} C_VEL
LIN {X 0,Y 336.046,Z 490.309,A -85,B 0,C 180,E1 -14668.651,E2 -14668.651} C_VEL
LIN {X 0,Y 335.078,Z 498.871,A -85,B 0,C 180,E1 -14669.999,E2 -14669.999} C_VEL
LIN {X 0,Y 334.196,Z 506.759,A -85,B 0,C 180,E1 -14671.505,E2 -14671.505} C_VEL
LIN {X 0,Y 333.438,Z 514.446,A -85,B 0,C 180,E1 -14673.322,E2 -14673.322} C_VEL
LIN {X 0,Y 332.841,Z 519.726,A -85,B 0,C 180,E1 -14674.844,E2 -14674.844} C_VEL
LIN {X 0,Y 332.552,Z 524.754,A -85,B 0,C 180,E1 -14676.65,E2 -14676.65} C_VEL
LIN {X 0,Y 332.204,Z 528.777,A -85,B 0,C 180,E1 -14678.515,E2 -14678.515} C_VEL
LIN {X 0,Y 332.008,Z 530.822,A -85,B 0,C 180,E1 -14679.749,E2 -14679.749} C_VEL
LIN {X 0,Y 331.888,Z 532.445,A -85,B 0,C 180,E1 -14680.986,E2 -14680.986} C_VEL
LIN {X 0,Y 331.853,Z 534.191,A -85,B 0,C 180,E1 -14683.047,E2 -14683.047} C_VEL
LIN {X 0,Y 331.803,Z 534.738,A -85,B 0,C 180,E1 -14684.723,E2 -14684.723} C_VEL
LIN {X 0,Y 331.817,Z 534.689,A -85,B 0,C 180,E1 -14685.981,E2 -14685.981} C_VEL
LIN {X 0,Y 332.031,Z 533.875,A -85,B 0,C 180,E1 -14687.731,E2 -14687.731} C_VEL
LIN {X 0,Y 332.332,Z 531.906,A -85,B 0,C 180,E1 -14689.776,E2 -14689.776} C_VEL
LIN {X 0,Y 332.879,Z 528.919,A -85,B 0,C 180,E1 -14691.727,E2 -14691.727} C_VEL
LIN {X 0,Y 333.528,Z 524.959,A -85,B 0,C 180,E1 -14693.599,E2 -14693.599} C_VEL
LIN {X 0,Y 334.533,Z 519.167,A -85,B 0,C 180,E1 -14695.667,E2 -14695.667} C_VEL
LIN {X 0,Y 335.834,Z 511.578,A -85,B 0,C 180,E1 -14697.749,E2 -14697.749} C_VEL
LIN {X 0,Y 337.071,Z 504.638,A -85,B 0,C 180,E1 -14699.269,E2 -14699.269} C_VEL
LIN {X 0,Y 338.55,Z 495.465,A -85,B 0,C 180,E1 -14700.915,E2 -14700.915} C_VEL
LIN {X 0,Y 340.044,Z 485.807,A -85,B 0,C 180,E1 -14702.299,E2 -14702.299} C_VEL
LIN {X 0,Y 341.586,Z 474.748,A -85,B 0,C 180,E1 -14703.568,E2 -14703.568} C_VEL
LIN {X 0,Y 342.998,Z 462.657,A -85,B 0,C 180,E1 -14704.651,E2 -14704.651} C_VEL
LIN {X 0,Y 344.183,Z 449.88,A -85,B 0,C 180,E1 -14705.496,E2 -14705.496} C_VEL
LIN {X 0,Y 345.03,Z 436.571,A -85,B 0,C 180,E1 -14706.115,E2 -14706.115} C_VEL
LIN {X 0,Y 345.587,Z 422.762,A -85,B 0,C 180,E1 -14706.487,E2 -14706.487} C_VEL
LIN {X 0,Y 345.884,Z 410.448,A -85,B 0,C 180,E1 -14706.747,E2 -14706.747} C_VEL
LIN {X 0,Y 345.436,Z 404.645,A -85,B 0,C 180,E1 -14706.919,E2 -14706.919} C_VEL
LIN {X 0,Y 340.807,Z 386.014,A -85,B 0,C 180,E1 -14707.761,E2 -14707.761} C_VEL
LIN {X 0,Y 340.441,Z 380.21,A -85,B 0,C 180,E1 -14707.932,E2 -14707.932} C_VEL
LIN {X 0,Y 341.053,Z 355.672,A -85,B 0,C 180,E1 -14708.459,E2 -14708.459} C_VEL
LIN {X 0,Y 338.81,Z 346.07,A -85,B 0,C 180,E1 -14708.898,E2 -14708.898} C_VEL
LIN {X 0,Y 331.836,Z 330.383,A -85,B 0,C 180,E1 -14709.967,E2 -14709.967} C_VEL
LIN {X 0,Y 328.884,Z 324.048,A -85,B 0,C 180,E1 -14710.452,E2 -14710.452} C_VEL
LIN {X 0,Y 326.576,Z 314.806,A -85,B 0,C 180,E1 -14713.521,E2 -14713.521} C_VEL
LIN {X 0,Y 326.566,Z 314.797,A -85,B 0,C 180,E1 -14717.028,E2 -14717.028} C_VEL
LIN {X 0,Y 326.574,Z 314.808,A -85,B 0,C 180,E1 -14721.385,E2 -14721.385} C_VEL
LIN {X 0,Y 326.611,Z 314.79,A -85,B 0,C 180,E1 -14724.851,E2 -14724.851} C_VEL
LIN {X 0,Y 326.6,Z 314.789,A -85,B 0,C 180,E1 -14727.455,E2 -14727.455} C_VEL
LIN {X 0,Y 326.608,Z 314.795,A -85,B 0,C 180,E1 -14730.336,E2 -14730.336} C_VEL
LIN {X 0,Y 326.594,Z 314.797,A -85,B 0,C 180,E1 -14734.509,E2 -14734.509} C_VEL
LIN {X 0,Y 326.601,Z 314.797,A -85,B 0,C 180,E1 -14738.542,E2 -14738.542} C_VEL
LIN {X 0,Y 326.639,Z 314.794,A -85,B 0,C 180,E1 -14741.206,E2 -14741.206} C_VEL
LIN {X 0,Y 326.716,Z 314.785,A -85,B 0,C 180,E1 -14745.459,E2 -14745.459} C_VEL
LIN {X 0,Y 326.745,Z 314.782,A -85,B 0,C 180,E1 -14748.838,E2 -14748.838} C_VEL
LIN {X 0,Y 326.901,Z 314.757,A -85,B 0,C 180,E1 -14752.589,E2 -14752.589} C_VEL
LIN {X 0,Y 326.732,Z 314.781,A -85,B 0,C 180,E1 -14755.064,E2 -14755.064} C_VEL
LIN {X 0,Y 326.975,Z 314.745,A -85,B 0,C 180,E1 -14757.537,E2 -14757.537} C_VEL
LIN {X 0,Y 327.035,Z 314.739,A -85,B 0,C 180,E1 -14761.232,E2 -14761.232} C_VEL
LIN {X 0,Y 326.728,Z 314.78,A -85,B 0,C 180,E1 -14763.7,E2 -14763.7} C_VEL
LIN {X 0,Y 326.942,Z 314.758,A -85,B 0,C 180,E1 -14766.17,E2 -14766.17} C_VEL
LIN {X 0,Y 326.774,Z 314.775,A -85,B 0,C 180,E1 -14769.908,E2 -14769.908} C_VEL
LIN {X 0,Y 326.751,Z 314.77,A -85,B 0,C 180,E1 -14773.686,E2 -14773.686} C_VEL
LIN {X 0,Y 326.656,Z 314.782,A -85,B 0,C 180,E1 -14777.531,E2 -14777.531} C_VEL
LIN {X 0,Y 326.64,Z 314.792,A -85,B 0,C 180,E1 -14780.137,E2 -14780.137} C_VEL
LIN {X 0,Y 326.604,Z 314.795,A -85,B 0,C 180,E1 -14784.133,E2 -14784.133} C_VEL
LIN {X 0,Y 326.592,Z 314.797,A -85,B 0,C 180,E1 -14788.257,E2 -14788.257} C_VEL
LIN {X 0,Y 326.567,Z 314.802,A -85,B 0,C 180,E1 -14791.098,E2 -14791.098} C_VEL
LIN {X 0,Y 326.601,Z 314.801,A -85,B 0,C 180,E1 -14794.02,E2 -14794.02} C_VEL
LIN {X 0,Y 326.617,Z 314.801,A -85,B 0,C 180,E1 -14797.239,E2 -14797.239} C_VEL
LIN {X 0,Y 326.54,Z 314.812,A -85,B 0,C 180,E1 -14801.126,E2 -14801.126} C_VEL
LIN {X 0,Y 326.556,Z 314.788,A -85,B 0,C 180,E1 -14803.527,E2 -14803.527} C_VEL
LIN {X 0,Y 326.572,Z 314.808,A -85,B 0,C 180,E1 -14807.029,E2 -14807.029} C_VEL
LIN {X 0,Y 326.607,Z 314.805,A -85,B 0,C 180,E1 -14810.774,E2 -14810.774} C_VEL
LIN {X 0,Y 326.61,Z 314.8,A -85,B 0,C 180,E1 -14814.482,E2 -14814.482} C_VEL
LIN {X 0,Y 326.649,Z 314.927,A -85,B 0,C 180,E1 -14816.198,E2 -14816.198} C_VEL
LIN {X 0,Y 329.518,Z 326.458,A -85,B 0,C 180,E1 -14819.921,E2 -14819.921} C_VEL
LIN {X 0,Y 331.598,Z 336.303,A -85,B 0,C 180,E1 -14822.894,E2 -14822.894} C_VEL
LIN {X 0,Y 332.19,Z 340.061,A -85,B 0,C 180,E1 -14823.97,E2 -14823.97} C_VEL
LIN {X 0,Y 334.227,Z 347.639,A -85,B 0,C 180,E1 -14824.359,E2 -14824.359} C_VEL
LIN {X 0,Y 339.145,Z 371.855,A -85,B 0,C 180,E1 -14825.412,E2 -14825.412} C_VEL
LIN {X 0,Y 340.463,Z 380.143,A -85,B 0,C 180,E1 -14825.73,E2 -14825.73} C_VEL
LIN {X 0,Y 338.701,Z 448.636,A -85,B 0,C 180,E1 -14827.226,E2 -14827.226} C_VEL
LIN {X 0,Y 337.784,Z 461.732,A -85,B 0,C 180,E1 -14827.726,E2 -14827.726} C_VEL
LIN {X 0,Y 336.675,Z 473.782,A -85,B 0,C 180,E1 -14828.414,E2 -14828.414} C_VEL
LIN {X 0,Y 335.346,Z 485.174,A -85,B 0,C 180,E1 -14829.29,E2 -14829.29} C_VEL
LIN {X 0,Y 333.596,Z 496.905,A -85,B 0,C 180,E1 -14830.463,E2 -14830.463} C_VEL
LIN {X 0,Y 331.887,Z 507.421,A -85,B 0,C 180,E1 -14831.801,E2 -14831.801} C_VEL
LIN {X 0,Y 330.354,Z 516.334,A -85,B 0,C 180,E1 -14833.205,E2 -14833.205} C_VEL
LIN {X 0,Y 329.062,Z 524.729,A -85,B 0,C 180,E1 -14834.834,E2 -14834.834} C_VEL
LIN {X 0,Y 327.599,Z 532.385,A -85,B 0,C 180,E1 -14836.668,E2 -14836.668} C_VEL
LIN {X 0,Y 326.414,Z 539.462,A -85,B 0,C 180,E1 -14838.828,E2 -14838.828} C_VEL
LIN {X 0,Y 325.681,Z 544.193,A -85,B 0,C 180,E1 -14840.687,E2 -14840.687} C_VEL
LIN {X 0,Y 325.2,Z 547.83,A -85,B 0,C 180,E1 -14842.551,E2 -14842.551} C_VEL
LIN {X 0,Y 324.984,Z 550.154,A -85,B 0,C 180,E1 -14844.146,E2 -14844.146} C_VEL
LIN {X 0,Y 324.876,Z 552.186,A -85,B 0,C 180,E1 -14846.28,E2 -14846.28} C_VEL
LIN {X 0,Y 324.833,Z 552.83,A -85,B 0,C 180,E1 -14847.521,E2 -14847.521} C_VEL
LIN {X 0,Y 324.821,Z 553.09,A -85,B 0,C 180,E1 -14848.761,E2 -14848.761} C_VEL
LIN {X 0,Y 324.876,Z 552.929,A -85,B 0,C 180,E1 -14850.001,E2 -14850.001} C_VEL
LIN {X 0,Y 324.839,Z 552.356,A -85,B 0,C 180,E1 -14851.241,E2 -14851.241} C_VEL
LIN {X 0,Y 324.847,Z 551.392,A -85,B 0,C 180,E1 -14852.481,E2 -14852.481} C_VEL
LIN {X 0,Y 324.906,Z 550.03,A -85,B 0,C 180,E1 -14853.722,E2 -14853.722} C_VEL
LIN {X 0,Y 324.988,Z 546.621,A -85,B 0,C 180,E1 -14855.86,E2 -14855.86} C_VEL
LIN {X 0,Y 325.237,Z 541.595,A -85,B 0,C 180,E1 -14858.075,E2 -14858.075} C_VEL
LIN {X 0,Y 325.657,Z 536.063,A -85,B 0,C 180,E1 -14859.943,E2 -14859.943} C_VEL
LIN {X 0,Y 326.315,Z 529.138,A -85,B 0,C 180,E1 -14861.807,E2 -14861.807} C_VEL
LIN {X 0,Y 327.129,Z 522.06,A -85,B 0,C 180,E1 -14863.354,E2 -14863.354} C_VEL
LIN {X 0,Y 328.123,Z 513.515,A -85,B 0,C 180,E1 -14864.895,E2 -14864.895} C_VEL
LIN {X 0,Y 329.073,Z 502.9,A -85,B 0,C 180,E1 -14866.439,E2 -14866.439} C_VEL
LIN {X 0,Y 330.215,Z 492.409,A -85,B 0,C 180,E1 -14867.656,E2 -14867.656} C_VEL
LIN {X 0,Y 331.293,Z 480.864,A -85,B 0,C 180,E1 -14868.716,E2 -14868.716} C_VEL
LIN {X 0,Y 332.249,Z 468.899,A -85,B 0,C 180,E1 -14869.542,E2 -14869.542} C_VEL
LIN {X 0,Y 333.063,Z 455.051,A -85,B 0,C 180,E1 -14870.215,E2 -14870.215} C_VEL
LIN {X 0,Y 333.523,Z 442.372,A -85,B 0,C 180,E1 -14870.589,E2 -14870.589} C_VEL
LIN {X 0,Y 334.573,Z 377.466,A -85,B 0,C 180,E1 -14871.98,E2 -14871.98} C_VEL
LIN {X 0,Y 329.383,Z 340.625,A -85,B 0,C 180,E1 -14873.126,E2 -14873.126} C_VEL
LIN {X 0,Y 330.081,Z 333.691,A -85,B 0,C 180,E1 -14874.868,E2 -14874.868} C_VEL
LIN {X 0,Y 328.635,Z 324.409,A -85,B 0,C 180,E1 -14877.374,E2 -14877.374} C_VEL
LIN {X 0,Y 326.663,Z 314.797,A -85,B 0,C 180,E1 -14880.119,E2 -14880.119} C_VEL
LIN {X 0,Y 326.611,Z 314.804,A -85,B 0,C 180,E1 -14884.02,E2 -14884.02} C_VEL
LIN {X 0,Y 326.627,Z 314.796,A -85,B 0,C 180,E1 -14887.238,E2 -14887.238} C_VEL
LIN {X 0,Y 326.548,Z 314.805,A -85,B 0,C 180,E1 -14891.125,E2 -14891.125} C_VEL
LIN {X 0,Y 326.565,Z 314.804,A -85,B 0,C 180,E1 -14893.526,E2 -14893.526} C_VEL
LIN {X 0,Y 326.579,Z 314.803,A -85,B 0,C 180,E1 -14897.029,E2 -14897.029} C_VEL
LIN {X 0,Y 326.615,Z 314.801,A -85,B 0,C 180,E1 -14900.773,E2 -14900.773} C_VEL
LIN {X 0,Y 326.617,Z 314.8,A -85,B 0,C 180,E1 -14904.481,E2 -14904.481} C_VEL
LIN {X 0,Y 326.612,Z 314.798,A -85,B 0,C 180,E1 -14907.456,E2 -14907.456} C_VEL
LIN {X 0,Y 326.629,Z 314.796,A -85,B 0,C 180,E1 -14910.337,E2 -14910.337} C_VEL
LIN {X 0,Y 326.632,Z 314.8,A -85,B 0,C 180,E1 -14913.137,E2 -14913.137} C_VEL
LIN {X 0,Y 326.648,Z 314.793,A -85,B 0,C 180,E1 -14915.87,E2 -14915.87} C_VEL
LIN {X 0,Y 326.628,Z 314.794,A -85,B 0,C 180,E1 -14919.862,E2 -14919.862} C_VEL
LIN {X 0,Y 326.713,Z 314.788,A -85,B 0,C 180,E1 -14923.761,E2 -14923.761} C_VEL
LIN {X 0,Y 326.764,Z 314.778,A -85,B 0,C 180,E1 -14926.315,E2 -14926.315} C_VEL
LIN {X 0,Y 326.808,Z 314.772,A -85,B 0,C 180,E1 -14930.093,E2 -14930.093} C_VEL
LIN {X 0,Y 326.965,Z 314.758,A -85,B 0,C 180,E1 -14933.83,E2 -14933.83} C_VEL
LIN {X 0,Y 327.02,Z 314.748,A -85,B 0,C 180,E1 -14937.536,E2 -14937.536} C_VEL
LIN {X 0,Y 327.162,Z 314.733,A -85,B 0,C 180,E1 -14940,E2 -14940} C_VEL
LIN {X 0,Y 327.038,Z 314.744,A -85,B 0,C 180,E1 -14942.463,E2 -14942.463} C_VEL
LIN {X 0,Y 326.924,Z 314.758,A -85,B 0,C 180,E1 -14946.517,E2 -14946.517} C_VEL
LIN {X 0,Y 326.787,Z 314.776,A -85,B 0,C 180,E1 -14949.907,E2 -14949.907} C_VEL
LIN {X 0,Y 326.763,Z 314.776,A -85,B 0,C 180,E1 -14953.685,E2 -14953.685} C_VEL
LIN {X 0,Y 326.667,Z 314.789,A -85,B 0,C 180,E1 -14957.529,E2 -14957.529} C_VEL
LIN {X 0,Y 326.622,Z 314.797,A -85,B 0,C 180,E1 -14961.456,E2 -14961.456} C_VEL
LIN {X 0,Y 326.647,Z 314.793,A -85,B 0,C 180,E1 -14965.487,E2 -14965.487} C_VEL
LIN {X 0,Y 326.631,Z 314.791,A -85,B 0,C 180,E1 -14968.253,E2 -14968.253} C_VEL
LIN {X 0,Y 326.578,Z 314.804,A -85,B 0,C 180,E1 -14971.096,E2 -14971.096} C_VEL
LIN {X 0,Y 326.61,Z 314.798,A -85,B 0,C 180,E1 -14974.019,E2 -14974.019} C_VEL
LIN {X 0,Y 326.631,Z 314.796,A -85,B 0,C 180,E1 -14977.238,E2 -14977.238} C_VEL
LIN {X 0,Y 326.579,Z 314.801,A -85,B 0,C 180,E1 -14981.13,E2 -14981.13} C_VEL
LIN {X 0,Y 326.529,Z 314.807,A -85,B 0,C 180,E1 -14984.742,E2 -14984.742} C_VEL
LIN {X 0,Y 326.576,Z 314.805,A -85,B 0,C 180,E1 -14988.153,E2 -14988.153} C_VEL
LIN {X 0,Y 326.588,Z 314.801,A -85,B 0,C 180,E1 -14991.385,E2 -14991.385} C_VEL
LIN {X 0,Y 326.621,Z 314.795,A -85,B 0,C 180,E1 -14994.851,E2 -14994.851} C_VEL
LIN {X 0,Y 326.611,Z 314.797,A -85,B 0,C 180,E1 -14997.455,E2 -14997.455} C_VEL
LIN {X 0,Y 326.626,Z 314.801,A -85,B 0,C 180,E1 -15000.336,E2 -15000.336} C_VEL
LIN {X 0,Y 326.63,Z 314.796,A -85,B 0,C 180,E1 -15003.136,E2 -15003.136} C_VEL
LIN {X 0,Y 326.647,Z 314.793,A -85,B 0,C 180,E1 -15005.87,E2 -15005.87} C_VEL
LIN {X 0,Y 326.658,Z 314.792,A -85,B 0,C 180,E1 -15009.864,E2 -15009.864} C_VEL
LIN {X 0,Y 326.665,Z 314.793,A -85,B 0,C 180,E1 -15012.469,E2 -15012.469} C_VEL
LIN {X 0,Y 326.76,Z 314.78,A -85,B 0,C 180,E1 -15016.314,E2 -15016.314} C_VEL
LIN {X 0,Y 326.798,Z 314.878,A -85,B 0,C 180,E1 -15018.289,E2 -15018.289} C_VEL
LIN {X 0,Y 328.527,Z 323.739,A -85,B 0,C 180,E1 -15020.901,E2 -15020.901} C_VEL
LIN {X 0,Y 331.309,Z 332.957,A -85,B 0,C 180,E1 -15021.288,E2 -15021.288} C_VEL
LIN {X 0,Y 335.088,Z 353.424,A -85,B 0,C 180,E1 -15021.969,E2 -15021.969} C_VEL
LIN {X 0,Y 333.46,Z 431.625,A -85,B 0,C 180,E1 -15023.662,E2 -15023.662} C_VEL
LIN {X 0,Y 332.933,Z 443.579,A -85,B 0,C 180,E1 -15024.13,E2 -15024.13} C_VEL
LIN {X 0,Y 332.183,Z 456.984,A -85,B 0,C 180,E1 -15024.916,E2 -15024.916} C_VEL
LIN {X 0,Y 331.312,Z 468.411,A -85,B 0,C 180,E1 -15025.83,E2 -15025.83} C_VEL
LIN {X 0,Y 330.313,Z 479.276,A -85,B 0,C 180,E1 -15026.95,E2 -15026.95} C_VEL
LIN {X 0,Y 329.172,Z 489.875,A -85,B 0,C 180,E1 -15028.317,E2 -15028.317} C_VEL
LIN {X 0,Y 328.18,Z 498.538,A -85,B 0,C 180,E1 -15029.692,E2 -15029.692} C_VEL
LIN {X 0,Y 327.259,Z 506.515,A -85,B 0,C 180,E1 -15031.229,E2 -15031.229} C_VEL
LIN {X 0,Y 326.424,Z 514.315,A -85,B 0,C 180,E1 -15033.084,E2 -15033.084} C_VEL
LIN {X 0,Y 325.744,Z 520.565,A -85,B 0,C 180,E1 -15034.95,E2 -15034.95} C_VEL
LIN {X 0,Y 325.456,Z 525.055,A -85,B 0,C 180,E1 -15036.62,E2 -15036.62} C_VEL
LIN {X 0,Y 325.069,Z 529.359,A -85,B 0,C 180,E1 -15038.703,E2 -15038.703} C_VEL
LIN {X 0,Y 324.878,Z 531.344,A -85,B 0,C 180,E1 -15039.965,E2 -15039.965} C_VEL
LIN {X 0,Y 324.788,Z 532.901,A -85,B 0,C 180,E1 -15041.229,E2 -15041.229} C_VEL
LIN {X 0,Y 324.755,Z 534.406,A -85,B 0,C 180,E1 -15043.135,E2 -15043.135} C_VEL
LIN {X 0,Y 324.696,Z 534.971,A -85,B 0,C 180,E1 -15045.053,E2 -15045.053} C_VEL
LIN {X 0,Y 324.752,Z 534.833,A -85,B 0,C 180,E1 -15046.339,E2 -15046.339} C_VEL
LIN {X 0,Y 324.976,Z 534.069,A -85,B 0,C 180,E1 -15047.908,E2 -15047.908} C_VEL
LIN {X 0,Y 325.338,Z 531.833,A -85,B 0,C 180,E1 -15050.219,E2 -15050.219} C_VEL
LIN {X 0,Y 325.849,Z 529.154,A -85,B 0,C 180,E1 -15051.962,E2 -15051.962} C_VEL
LIN {X 0,Y 326.666,Z 524.6,A -85,B 0,C 180,E1 -15054.126,E2 -15054.126} C_VEL
LIN {X 0,Y 327.892,Z 518.111,A -85,B 0,C 180,E1 -15056.391,E2 -15056.391} C_VEL
LIN {X 0,Y 329.214,Z 510.973,A -85,B 0,C 180,E1 -15058.327,E2 -15058.327} C_VEL
LIN {X 0,Y 330.569,Z 503.38,A -85,B 0,C 180,E1 -15059.973,E2 -15059.973} C_VEL
LIN {X 0,Y 332.141,Z 494.221,A -85,B 0,C 180,E1 -15061.579,E2 -15061.579} C_VEL
LIN {X 0,Y 333.664,Z 484.756,A -85,B 0,C 180,E1 -15062.924,E2 -15062.924} C_VEL
LIN {X 0,Y 335.181,Z 474.356,A -85,B 0,C 180,E1 -15064.116,E2 -15064.116} C_VEL
LIN {X 0,Y 336.631,Z 462.236,A -85,B 0,C 180,E1 -15065.203,E2 -15065.203} C_VEL
LIN {X 0,Y 337.865,Z 449.003,A -85,B 0,C 180,E1 -15066.08,E2 -15066.08} C_VEL
LIN {X 0,Y 338.716,Z 436.201,A -85,B 0,C 180,E1 -15066.667,E2 -15066.667} C_VEL
LIN {X 0,Y 339.305,Z 420.906,A -85,B 0,C 180,E1 -15067.069,E2 -15067.069} C_VEL
LIN {X 0,Y 340.441,Z 380.21,A -85,B 0,C 180,E1 -15067.932,E2 -15067.932} C_VEL
LIN {X 0,Y 340.142,Z 374.386,A -85,B 0,C 180,E1 -15068.098,E2 -15068.098} C_VEL
LIN {X 0,Y 338.998,Z 368.731,A -85,B 0,C 180,E1 -15068.338,E2 -15068.338} C_VEL
LIN {X 0,Y 333.442,Z 350.3,A -85,B 0,C 180,E1 -15069.314,E2 -15069.314} C_VEL
LIN {X 0,Y 326.809,Z 334.862,A -85,B 0,C 180,E1 -15070.375,E2 -15070.375} C_VEL
LIN {X 0,Y 321.693,Z 324.226,A -85,B 0,C 180,E1 -15071.237,E2 -15071.237} C_VEL
LIN {X 0,Y 319.5,Z 315.69,A -85,B 0,C 180,E1 -15074.223,E2 -15074.223} C_VEL
LIN {X 0,Y 319.545,Z 315.672,A -85,B 0,C 180,E1 -15077.015,E2 -15077.015} C_VEL
LIN {X 0,Y 319.537,Z 315.681,A -85,B 0,C 180,E1 -15080.37,E2 -15080.37} C_VEL
LIN {X 0,Y 319.572,Z 315.674,A -85,B 0,C 180,E1 -15084.457,E2 -15084.457} C_VEL
LIN {X 0,Y 319.516,Z 315.682,A -85,B 0,C 180,E1 -15088.137,E2 -15088.137} C_VEL
LIN {X 0,Y 319.563,Z 315.677,A -85,B 0,C 180,E1 -15091.603,E2 -15091.603} C_VEL
LIN {X 0,Y 319.541,Z 315.679,A -85,B 0,C 180,E1 -15095.299,E2 -15095.299} C_VEL
LIN {X 0,Y 319.554,Z 315.673,A -85,B 0,C 180,E1 -15098.045,E2 -15098.045} C_VEL
LIN {X 0,Y 319.577,Z 315.668,A -85,B 0,C 180,E1 -15102.069,E2 -15102.069} C_VEL
LIN {X 0,Y 319.7,Z 315.652,A -85,B 0,C 180,E1 -15106.007,E2 -15106.007} C_VEL
LIN {X 0,Y 319.724,Z 315.656,A -85,B 0,C 180,E1 -15109.872,E2 -15109.872} C_VEL
LIN {X 0,Y 319.886,Z 315.635,A -85,B 0,C 180,E1 -15113.694,E2 -15113.694} C_VEL
LIN {X 0,Y 319.985,Z 315.627,A -85,B 0,C 180,E1 -15118.742,E2 -15118.742} C_VEL
LIN {X 0,Y 320.002,Z 315.615,A -85,B 0,C 180,E1 -15121.259,E2 -15121.259} C_VEL
LIN {X 0,Y 319.898,Z 315.632,A -85,B 0,C 180,E1 -15126.307,E2 -15126.307} C_VEL
LIN {X 0,Y 319.726,Z 315.654,A -85,B 0,C 180,E1 -15130.128,E2 -15130.128} C_VEL
LIN {X 0,Y 319.724,Z 315.646,A -85,B 0,C 180,E1 -15133.993,E2 -15133.993} C_VEL
LIN {X 0,Y 319.617,Z 315.657,A -85,B 0,C 180,E1 -15137.93,E2 -15137.93} C_VEL
LIN {X 0,Y 319.588,Z 315.672,A -85,B 0,C 180,E1 -15140.601,E2 -15140.601} C_VEL
LIN {X 0,Y 319.535,Z 315.671,A -85,B 0,C 180,E1 -15143.322,E2 -15143.322} C_VEL
LIN {X 0,Y 319.546,Z 315.677,A -85,B 0,C 180,E1 -15146.096,E2 -15146.096} C_VEL
LIN {X 0,Y 319.537,Z 315.678,A -85,B 0,C 180,E1 -15148.939,E2 -15148.939} C_VEL
LIN {X 0,Y 319.518,Z 315.677,A -85,B 0,C 180,E1 -15151.864,E2 -15151.864} C_VEL
LIN {X 0,Y 319.573,Z 315.672,A -85,B 0,C 180,E1 -15155.544,E2 -15155.544} C_VEL
LIN {X 0,Y 319.522,Z 315.681,A -85,B 0,C 180,E1 -15159.663,E2 -15159.663} C_VEL
LIN {X 0,Y 319.515,Z 315.664,A -85,B 0,C 180,E1 -15163.462,E2 -15163.462} C_VEL
LIN {X 0,Y 319.55,Z 315.683,A -85,B 0,C 180,E1 -15167.018,E2 -15167.018} C_VEL
LIN {X 0,Y 319.543,Z 315.686,A -85,B 0,C 180,E1 -15170.372,E2 -15170.372} C_VEL
LIN {X 0,Y 319.577,Z 315.676,A -85,B 0,C 180,E1 -15174.458,E2 -15174.458} C_VEL
LIN {X 0,Y 319.583,Z 315.715,A -85,B 0,C 180,E1 -15175.511,E2 -15175.511} C_VEL
LIN {X 0,Y 322.344,Z 326.692,A -85,B 0,C 180,E1 -15179.18,E2 -15179.18} C_VEL
LIN {X 0,Y 324.694,Z 337.529,A -85,B 0,C 180,E1 -15182.555,E2 -15182.555} C_VEL
LIN {X 0,Y 325.153,Z 340.007,A -85,B 0,C 180,E1 -15183.243,E2 -15183.243} C_VEL
LIN {X 0,Y 327.574,Z 346.793,A -85,B 0,C 180,E1 -15183.669,E2 -15183.669} C_VEL
LIN {X 0,Y 332.768,Z 372.005,A -85,B 0,C 180,E1 -15184.815,E2 -15184.815} C_VEL
LIN {X 0,Y 334.185,Z 380.775,A -85,B 0,C 180,E1 -15185.164,E2 -15185.164} C_VEL
LIN {X 0,Y 332.368,Z 448.853,A -85,B 0,C 180,E1 -15186.685,E2 -15186.685} C_VEL
LIN {X 0,Y 331.428,Z 461.809,A -85,B 0,C 180,E1 -15187.193,E2 -15187.193} C_VEL
LIN {X 0,Y 330.244,Z 473.793,A -85,B 0,C 180,E1 -15187.89,E2 -15187.89} C_VEL
LIN {X 0,Y 328.946,Z 484.268,A -85,B 0,C 180,E1 -15188.704,E2 -15188.704} C_VEL
LIN {X 0,Y 327.41,Z 494.867,A -85,B 0,C 180,E1 -15189.751,E2 -15189.751} C_VEL
LIN {X 0,Y 325.556,Z 505.725,A -85,B 0,C 180,E1 -15191.108,E2 -15191.108} C_VEL
LIN {X 0,Y 323.787,Z 515.423,A -85,B 0,C 180,E1 -15192.627,E2 -15192.627} C_VEL
LIN {X 0,Y 322.478,Z 523.48,A -85,B 0,C 180,E1 -15194.193,E2 -15194.193} C_VEL
LIN {X 0,Y 320.935,Z 531.373,A -85,B 0,C 180,E1 -15196.063,E2 -15196.063} C_VEL
LIN {X 0,Y 319.74,Z 537.703,A -85,B 0,C 180,E1 -15197.948,E2 -15197.948} C_VEL
LIN {X 0,Y 318.875,Z 542.761,A -85,B 0,C 180,E1 -15199.846,E2 -15199.846} C_VEL
LIN {X 0,Y 318.285,Z 546.706,A -85,B 0,C 180,E1 -15201.749,E2 -15201.749} C_VEL
LIN {X 0,Y 317.871,Z 550.305,A -85,B 0,C 180,E1 -15204.232,E2 -15204.232} C_VEL
LIN {X 0,Y 317.786,Z 552.042,A -85,B 0,C 180,E1 -15206.197,E2 -15206.197} C_VEL
LIN {X 0,Y 317.754,Z 552.665,A -85,B 0,C 180,E1 -15207.466,E2 -15207.466} C_VEL
LIN {X 0,Y 317.733,Z 552.896,A -85,B 0,C 180,E1 -15208.734,E2 -15208.734} C_VEL
LIN {X 0,Y 317.783,Z 552.697,A -85,B 0,C 180,E1 -15210.001,E2 -15210.001} C_VEL
LIN {X 0,Y 317.75,Z 552.101,A -85,B 0,C 180,E1 -15211.269,E2 -15211.269} C_VEL
LIN {X 0,Y 317.768,Z 551.115,A -85,B 0,C 180,E1 -15212.536,E2 -15212.536} C_VEL
LIN {X 0,Y 317.815,Z 549.724,A -85,B 0,C 180,E1 -15213.805,E2 -15213.805} C_VEL
LIN {X 0,Y 317.882,Z 546.645,A -85,B 0,C 180,E1 -15215.786,E2 -15215.786} C_VEL
LIN {X 0,Y 318.065,Z 542.778,A -85,B 0,C 180,E1 -15217.62,E2 -15217.62} C_VEL
LIN {X 0,Y 318.536,Z 536.599,A -85,B 0,C 180,E1 -15219.847,E2 -15219.847} C_VEL
LIN {X 0,Y 319.188,Z 529.837,A -85,B 0,C 180,E1 -15221.753,E2 -15221.753} C_VEL
LIN {X 0,Y 320.164,Z 521.436,A -85,B 0,C 180,E1 -15223.65,E2 -15223.65} C_VEL
LIN {X 0,Y 321.218,Z 512.77,A -85,B 0,C 180,E1 -15225.223,E2 -15225.223} C_VEL
LIN {X 0,Y 322.222,Z 502.036,A -85,B 0,C 180,E1 -15226.799,E2 -15226.799} C_VEL
LIN {X 0,Y 323.377,Z 491.398,A -85,B 0,C 180,E1 -15228.042,E2 -15228.042} C_VEL
LIN {X 0,Y 324.547,Z 479.564,A -85,B 0,C 180,E1 -15229.12,E2 -15229.12} C_VEL
LIN {X 0,Y 325.528,Z 467.232,A -85,B 0,C 180,E1 -15229.962,E2 -15229.962} C_VEL
LIN {X 0,Y 326.334,Z 453.678,A -85,B 0,C 180,E1 -15230.61,E2 -15230.61} C_VEL
LIN {X 0,Y 326.819,Z 438.154,A -85,B 0,C 180,E1 -15231.031,E2 -15231.031} C_VEL
LIN {X 0,Y 327.814,Z 378.171,A -85,B 0,C 180,E1 -15232.344,E2 -15232.344} C_VEL
LIN {X 0,Y 322.544,Z 340.366,A -85,B 0,C 180,E1 -15233.562,E2 -15233.562} C_VEL
LIN {X 0,Y 323.086,Z 334.393,A -85,B 0,C 180,E1 -15235.1,E2 -15235.1} C_VEL
LIN {X 0,Y 321.297,Z 323.759,A -85,B 0,C 180,E1 -15238.054,E2 -15238.054} C_VEL
LIN {X 0,Y 319.627,Z 315.672,A -85,B 0,C 180,E1 -15240.45,E2 -15240.45} C_VEL
LIN {X 0,Y 319.581,Z 315.674,A -85,B 0,C 180,E1 -15243.353,E2 -15243.353} C_VEL
LIN {X 0,Y 319.56,Z 315.679,A -85,B 0,C 180,E1 -15246.428,E2 -15246.428} C_VEL
LIN {X 0,Y 319.532,Z 315.681,A -85,B 0,C 180,E1 -15249.662,E2 -15249.662} C_VEL
LIN {X 0,Y 319.525,Z 315.681,A -85,B 0,C 180,E1 -15253.461,E2 -15253.461} C_VEL
LIN {X 0,Y 319.558,Z 315.678,A -85,B 0,C 180,E1 -15257.017,E2 -15257.017} C_VEL
LIN {X 0,Y 319.551,Z 315.681,A -85,B 0,C 180,E1 -15260.371,E2 -15260.371} C_VEL
LIN {X 0,Y 319.585,Z 315.676,A -85,B 0,C 180,E1 -15264.457,E2 -15264.457} C_VEL
LIN {X 0,Y 319.529,Z 315.68,A -85,B 0,C 180,E1 -15268.138,E2 -15268.138} C_VEL
LIN {X 0,Y 319.598,Z 315.672,A -85,B 0,C 180,E1 -15271.596,E2 -15271.596} C_VEL
LIN {X 0,Y 319.588,Z 315.677,A -85,B 0,C 180,E1 -15275.302,E2 -15275.302} C_VEL
LIN {X 0,Y 319.572,Z 315.673,A -85,B 0,C 180,E1 -15278.046,E2 -15278.046} C_VEL
LIN {X 0,Y 319.618,Z 315.668,A -85,B 0,C 180,E1 -15282.07,E2 -15282.07} C_VEL
LIN {X 0,Y 319.737,Z 315.655,A -85,B 0,C 180,E1 -15286.008,E2 -15286.008} C_VEL
LIN {X 0,Y 319.756,Z 315.651,A -85,B 0,C 180,E1 -15289.872,E2 -15289.872} C_VEL
LIN {X 0,Y 319.922,Z 315.633,A -85,B 0,C 180,E1 -15293.694,E2 -15293.694} C_VEL
LIN {X 0,Y 319.966,Z 315.626,A -85,B 0,C 180,E1 -15297.482,E2 -15297.482} C_VEL
LIN {X 0,Y 320.115,Z 315.61,A -85,B 0,C 180,E1 -15300,E2 -15300} C_VEL
LIN {X 0,Y 319.982,Z 315.622,A -85,B 0,C 180,E1 -15302.517,E2 -15302.517} C_VEL
LIN {X 0,Y 319.888,Z 315.637,A -85,B 0,C 180,E1 -15306.499,E2 -15306.499} C_VEL
LIN {X 0,Y 319.739,Z 315.656,A -85,B 0,C 180,E1 -15310.127,E2 -15310.127} C_VEL
LIN {X 0,Y 319.736,Z 315.651,A -85,B 0,C 180,E1 -15313.992,E2 -15313.992} C_VEL
LIN {X 0,Y 319.617,Z 315.666,A -85,B 0,C 180,E1 -15317.929,E2 -15317.929} C_VEL
LIN {X 0,Y 319.571,Z 315.674,A -85,B 0,C 180,E1 -15321.954,E2 -15321.954} C_VEL
LIN {X 0,Y 319.582,Z 315.67,A -85,B 0,C 180,E1 -15326.092,E2 -15326.092} C_VEL
LIN {X 0,Y 319.561,Z 315.674,A -85,B 0,C 180,E1 -15328.936,E2 -15328.936} C_VEL
LIN {X 0,Y 319.528,Z 315.68,A -85,B 0,C 180,E1 -15331.862,E2 -15331.862} C_VEL
LIN {X 0,Y 319.583,Z 315.676,A -85,B 0,C 180,E1 -15335.542,E2 -15335.542} C_VEL
LIN {X 0,Y 319.561,Z 315.678,A -85,B 0,C 180,E1 -15339.668,E2 -15339.668} C_VEL
LIN {X 0,Y 319.523,Z 315.683,A -85,B 0,C 180,E1 -15343.46,E2 -15343.46} C_VEL
LIN {X 0,Y 319.555,Z 315.674,A -85,B 0,C 180,E1 -15347.016,E2 -15347.016} C_VEL
LIN {X 0,Y 319.547,Z 315.68,A -85,B 0,C 180,E1 -15350.37,E2 -15350.37} C_VEL
LIN {X 0,Y 319.581,Z 315.674,A -85,B 0,C 180,E1 -15354.456,E2 -15354.456} C_VEL
LIN {X 0,Y 319.527,Z 315.684,A -85,B 0,C 180,E1 -15358.137,E2 -15358.137} C_VEL
LIN {X 0,Y 319.595,Z 315.671,A -85,B 0,C 180,E1 -15361.595,E2 -15361.595} C_VEL
LIN {X 0,Y 319.586,Z 315.673,A -85,B 0,C 180,E1 -15365.301,E2 -15365.301} C_VEL
LIN {X 0,Y 319.599,Z 315.672,A -85,B 0,C 180,E1 -15368.047,E2 -15368.047} C_VEL
LIN {X 0,Y 319.659,Z 315.669,A -85,B 0,C 180,E1 -15370.978,E2 -15370.978} C_VEL
LIN {X 0,Y 319.713,Z 315.661,A -85,B 0,C 180,E1 -15375.288,E2 -15375.288} C_VEL
LIN {X 0,Y 319.734,Z 315.74,A -85,B 0,C 180,E1 -15377.986,E2 -15377.986} C_VEL
LIN {X 0,Y 321.452,Z 324.206,A -85,B 0,C 180,E1 -15380.486,E2 -15380.486} C_VEL
LIN {X 0,Y 324.842,Z 335.209,A -85,B 0,C 180,E1 -15380.953,E2 -15380.953} C_VEL
LIN {X 0,Y 328.317,Z 354.38,A -85,B 0,C 180,E1 -15381.601,E2 -15381.601} C_VEL
LIN {X 0,Y 326.65,Z 432.072,A -85,B 0,C 180,E1 -15383.319,E2 -15383.319} C_VEL
LIN {X 0,Y 326.119,Z 444.246,A -85,B 0,C 180,E1 -15383.813,E2 -15383.813} C_VEL
LIN {X 0,Y 325.356,Z 456.983,A -85,B 0,C 180,E1 -15384.576,E2 -15384.576} C_VEL
LIN {X 0,Y 324.501,Z 467.95,A -85,B 0,C 180,E1 -15385.461,E2 -15385.461} C_VEL
LIN {X 0,Y 323.364,Z 480.003,A -85,B 0,C 180,E1 -15386.728,E2 -15386.728} C_VEL
LIN {X 0,Y 322.173,Z 490.516,A -85,B 0,C 180,E1 -15388.124,E2 -15388.124} C_VEL
LIN {X 0,Y 321.043,Z 499.985,A -85,B 0,C 180,E1 -15389.685,E2 -15389.685} C_VEL
LIN {X 0,Y 319.965,Z 509.092,A -85,B 0,C 180,E1 -15391.572,E2 -15391.572} C_VEL
LIN {X 0,Y 319.159,Z 516.431,A -85,B 0,C 180,E1 -15393.471,E2 -15393.471} C_VEL
LIN {X 0,Y 318.65,Z 521.403,A -85,B 0,C 180,E1 -15395.06,E2 -15395.06} C_VEL
LIN {X 0,Y 318.313,Z 526.081,A -85,B 0,C 180,E1 -15396.91,E2 -15396.91} C_VEL
LIN {X 0,Y 317.956,Z 529.94,A -85,B 0,C 180,E1 -15398.9,E2 -15398.9} C_VEL
LIN {X 0,Y 317.753,Z 531.866,A -85,B 0,C 180,E1 -15400.19,E2 -15400.19} C_VEL
LIN {X 0,Y 317.698,Z 533.31,A -85,B 0,C 180,E1 -15401.483,E2 -15401.483} C_VEL
LIN {X 0,Y 317.652,Z 534.617,A -85,B 0,C 180,E1 -15403.223,E2 -15403.223} C_VEL
LIN {X 0,Y 317.626,Z 535.185,A -85,B 0,C 180,E1 -15405.397,E2 -15405.397} C_VEL
LIN {X 0,Y 317.711,Z 534.948,A -85,B 0,C 180,E1 -15406.711,E2 -15406.711} C_VEL
LIN {X 0,Y 317.924,Z 534.263,A -85,B 0,C 180,E1 -15408.094,E2 -15408.094} C_VEL
LIN {X 0,Y 318.076,Z 533.25,A -85,B 0,C 180,E1 -15409.354,E2 -15409.354} C_VEL
LIN {X 0,Y 318.367,Z 531.711,A -85,B 0,C 180,E1 -15410.682,E2 -15410.682} C_VEL
LIN {X 0,Y 319.03,Z 528.485,A -85,B 0,C 180,E1 -15412.704,E2 -15412.704} C_VEL
LIN {X 0,Y 319.846,Z 524.208,A -85,B 0,C 180,E1 -15414.675,E2 -15414.675} C_VEL
LIN {X 0,Y 320.967,Z 518.578,A -85,B 0,C 180,E1 -15416.67,E2 -15416.67} C_VEL
LIN {X 0,Y 322.383,Z 511.453,A -85,B 0,C 180,E1 -15418.658,E2 -15418.658} C_VEL
LIN {X 0,Y 323.774,Z 504.087,A -85,B 0,C 180,E1 -15420.308,E2 -15420.308} C_VEL
LIN {X 0,Y 325.423,Z 495.049,A -85,B 0,C 180,E1 -15421.944,E2 -15421.944} C_VEL
LIN {X 0,Y 327.207,Z 484.586,A -85,B 0,C 180,E1 -15423.46,E2 -15423.46} C_VEL
LIN {X 0,Y 328.802,Z 473.984,A -85,B 0,C 180,E1 -15424.686,E2 -15424.686} C_VEL
LIN {X 0,Y 330.172,Z 462.94,A -85,B 0,C 180,E1 -15425.692,E2 -15425.692} C_VEL
LIN {X 0,Y 331.409,Z 450.916,A -85,B 0,C 180,E1 -15426.518,E2 -15426.518} C_VEL
LIN {X 0,Y 332.305,Z 437.882,A -85,B 0,C 180,E1 -15427.161,E2 -15427.161} C_VEL
LIN {X 0,Y 332.94,Z 424.448,A -85,B 0,C 180,E1 -15427.553,E2 -15427.553} C_VEL
LIN {X 0,Y 334.766,Z 356.421,A -85,B 0,C 180,E1 -15429.035,E2 -15429.035} C_VEL
LIN {X 0,Y 333.442,Z 350.3,A -85,B 0,C 180,E1 -15429.314,E2 -15429.314} C_VEL
LIN {X 0,Y 332.225,Z 346.814,A -85,B 0,C 180,E1 -15429.52,E2 -15429.52} C_VEL
LIN {X 0,Y 329.321,Z 342.283,A -85,B 0,C 180,E1 -15429.927,E2 -15429.927} C_VEL
LIN {X 0,Y 318.121,Z 330.76,A -85,B 0,C 180,E1 -15431.429,E2 -15431.429} C_VEL
LIN {X 0,Y 316.025,Z 327.77,A -85,B 0,C 180,E1 -15431.748,E2 -15431.748} C_VEL
LIN {X 0,Y 314.482,Z 324.559,A -85,B 0,C 180,E1 -15432.026,E2 -15432.026} C_VEL
LIN {X 0,Y 312.455,Z 316.564,A -85,B 0,C 180,E1 -15434.909,E2 -15434.909} C_VEL
LIN {X 0,Y 312.448,Z 316.557,A -85,B 0,C 180,E1 -15437.924,E2 -15437.924} C_VEL
LIN {X 0,Y 312.476,Z 316.56,A -85,B 0,C 180,E1 -15441.922,E2 -15441.922} C_VEL
LIN {X 0,Y 312.523,Z 316.556,A -85,B 0,C 180,E1 -15444.22,E2 -15444.22} C_VEL
LIN {X 0,Y 312.493,Z 316.543,A -85,B 0,C 180,E1 -15447.333,E2 -15447.333} C_VEL
LIN {X 0,Y 312.498,Z 316.554,A -85,B 0,C 180,E1 -15451.291,E2 -15451.291} C_VEL
LIN {X 0,Y 312.516,Z 316.551,A -85,B 0,C 180,E1 -15454.705,E2 -15454.705} C_VEL
LIN {X 0,Y 312.531,Z 316.548,A -85,B 0,C 180,E1 -15457.525,E2 -15457.525} C_VEL
LIN {X 0,Y 312.542,Z 316.545,A -85,B 0,C 180,E1 -15461.651,E2 -15461.651} C_VEL
LIN {X 0,Y 312.642,Z 316.534,A -85,B 0,C 180,E1 -15465.684,E2 -15465.684} C_VEL
LIN {X 0,Y 312.674,Z 316.536,A -85,B 0,C 180,E1 -15469.641,E2 -15469.641} C_VEL
LIN {X 0,Y 312.785,Z 316.511,A -85,B 0,C 180,E1 -15472.252,E2 -15472.252} C_VEL
LIN {X 0,Y 312.673,Z 316.533,A -85,B 0,C 180,E1 -15474.842,E2 -15474.842} C_VEL
LIN {X 0,Y 312.953,Z 316.502,A -85,B 0,C 180,E1 -15478.714,E2 -15478.714} C_VEL
LIN {X 0,Y 312.969,Z 316.491,A -85,B 0,C 180,E1 -15481.287,E2 -15481.287} C_VEL
LIN {X 0,Y 312.839,Z 316.509,A -85,B 0,C 180,E1 -15486.45,E2 -15486.45} C_VEL
LIN {X 0,Y 312.742,Z 316.519,A -85,B 0,C 180,E1 -15489.051,E2 -15489.051} C_VEL
LIN {X 0,Y 312.625,Z 316.528,A -85,B 0,C 180,E1 -15492.992,E2 -15492.992} C_VEL
LIN {X 0,Y 312.614,Z 316.54,A -85,B 0,C 180,E1 -15495.651,E2 -15495.651} C_VEL
LIN {X 0,Y 312.556,Z 316.547,A -85,B 0,C 180,E1 -15499.712,E2 -15499.712} C_VEL
LIN {X 0,Y 312.51,Z 316.546,A -85,B 0,C 180,E1 -15502.777,E2 -15502.777} C_VEL
LIN {X 0,Y 312.479,Z 316.556,A -85,B 0,C 180,E1 -15506.733,E2 -15506.733} C_VEL
LIN {X 0,Y 312.49,Z 316.561,A -85,B 0,C 180,E1 -15509.656,E2 -15509.656} C_VEL
LIN {X 0,Y 312.514,Z 316.558,A -85,B 0,C 180,E1 -15513.69,E2 -15513.69} C_VEL
LIN {X 0,Y 312.505,Z 316.56,A -85,B 0,C 180,E1 -15517.388,E2 -15517.388} C_VEL
LIN {X 0,Y 312.436,Z 316.568,A -85,B 0,C 180,E1 -15520.718,E2 -15520.718} C_VEL
LIN {X 0,Y 312.446,Z 316.548,A -85,B 0,C 180,E1 -15524.211,E2 -15524.211} C_VEL
LIN {X 0,Y 312.48,Z 316.564,A -85,B 0,C 180,E1 -15527.92,E2 -15527.92} C_VEL
LIN {X 0,Y 312.495,Z 316.563,A -85,B 0,C 180,E1 -15530.972,E2 -15530.972} C_VEL
LIN {X 0,Y 312.55,Z 316.61,A -85,B 0,C 180,E1 -15534.818,E2 -15534.818} C_VEL
LIN {X 0,Y 314.862,Z 325.821,A -85,B 0,C 180,E1 -15538.016,E2 -15538.016} C_VEL
LIN {X 0,Y 317.123,Z 335.515,A -85,B 0,C 180,E1 -15541.185,E2 -15541.185} C_VEL
LIN {X 0,Y 317.967,Z 339.639,A -85,B 0,C 180,E1 -15542.45,E2 -15542.45} C_VEL
LIN {X 0,Y 321.577,Z 348.793,A -85,B 0,C 180,E1 -15543.086,E2 -15543.086} C_VEL
LIN {X 0,Y 326.544,Z 372.844,A -85,B 0,C 180,E1 -15544.22,E2 -15544.22} C_VEL
LIN {X 0,Y 328.001,Z 382.319,A -85,B 0,C 180,E1 -15544.604,E2 -15544.604} C_VEL
LIN {X 0,Y 326.074,Z 449.067,A -85,B 0,C 180,E1 -15546.123,E2 -15546.123} C_VEL
LIN {X 0,Y 325.104,Z 461.885,A -85,B 0,C 180,E1 -15546.639,E2 -15546.639} C_VEL
LIN {X 0,Y 323.83,Z 473.806,A -85,B 0,C 180,E1 -15547.344,E2 -15547.344} C_VEL
LIN {X 0,Y 322.392,Z 485.094,A -85,B 0,C 180,E1 -15548.249,E2 -15548.249} C_VEL
LIN {X 0,Y 320.546,Z 496.743,A -85,B 0,C 180,E1 -15549.465,E2 -15549.465} C_VEL
LIN {X 0,Y 318.692,Z 507.219,A -85,B 0,C 180,E1 -15550.852,E2 -15550.852} C_VEL
LIN {X 0,Y 316.803,Z 516.958,A -85,B 0,C 180,E1 -15552.461,E2 -15552.461} C_VEL
LIN {X 0,Y 315.395,Z 525.139,A -85,B 0,C 180,E1 -15554.16,E2 -15554.16} C_VEL
LIN {X 0,Y 313.806,Z 532.633,A -85,B 0,C 180,E1 -15556.07,E2 -15556.07} C_VEL
LIN {X 0,Y 312.462,Z 539.583,A -85,B 0,C 180,E1 -15558.322,E2 -15558.322} C_VEL
LIN {X 0,Y 311.643,Z 544.2,A -85,B 0,C 180,E1 -15560.264,E2 -15560.264} C_VEL
LIN {X 0,Y 311.076,Z 547.731,A -85,B 0,C 180,E1 -15562.211,E2 -15562.211} C_VEL
LIN {X 0,Y 310.766,Z 550.443,A -85,B 0,C 180,E1 -15564.307,E2 -15564.307} C_VEL
LIN {X 0,Y 310.7,Z 551.899,A -85,B 0,C 180,E1 -15566.11,E2 -15566.11} C_VEL
LIN {X 0,Y 310.677,Z 552.499,A -85,B 0,C 180,E1 -15567.408,E2 -15567.408} C_VEL
LIN {X 0,Y 310.648,Z 552.692,A -85,B 0,C 180,E1 -15568.705,E2 -15568.705} C_VEL
LIN {X 0,Y 310.693,Z 552.464,A -85,B 0,C 180,E1 -15570.001,E2 -15570.001} C_VEL
LIN {X 0,Y 310.664,Z 551.846,A -85,B 0,C 180,E1 -15571.297,E2 -15571.297} C_VEL
LIN {X 0,Y 310.691,Z 550.838,A -85,B 0,C 180,E1 -15572.594,E2 -15572.594} C_VEL
LIN {X 0,Y 310.727,Z 549.406,A -85,B 0,C 180,E1 -15573.892,E2 -15573.892} C_VEL
LIN {X 0,Y 310.778,Z 546.644,A -85,B 0,C 180,E1 -15575.713,E2 -15575.713} C_VEL
LIN {X 0,Y 311.007,Z 542.369,A -85,B 0,C 180,E1 -15577.794,E2 -15577.794} C_VEL
LIN {X 0,Y 311.508,Z 536.116,A -85,B 0,C 180,E1 -15580.071,E2 -15580.071} C_VEL
LIN {X 0,Y 312.201,Z 529.288,A -85,B 0,C 180,E1 -15582.02,E2 -15582.02} C_VEL
LIN {X 0,Y 313.191,Z 520.782,A -85,B 0,C 180,E1 -15583.96,E2 -15583.96} C_VEL
LIN {X 0,Y 314.292,Z 512.003,A -85,B 0,C 180,E1 -15585.566,E2 -15585.566} C_VEL
LIN {X 0,Y 315.354,Z 501.148,A -85,B 0,C 180,E1 -15587.176,E2 -15587.176} C_VEL
LIN {X 0,Y 316.578,Z 490.341,A -85,B 0,C 180,E1 -15588.443,E2 -15588.443} C_VEL
LIN {X 0,Y 317.798,Z 478.19,A -85,B 0,C 180,E1 -15589.542,E2 -15589.542} C_VEL
LIN {X 0,Y 318.806,Z 465.49,A -85,B 0,C 180,E1 -15590.402,E2 -15590.402} C_VEL
LIN {X 0,Y 319.559,Z 453.091,A -85,B 0,C 180,E1 -15590.983,E2 -15590.983} C_VEL
LIN {X 0,Y 320.08,Z 437.322,A -85,B 0,C 180,E1 -15591.411,E2 -15591.411} C_VEL
LIN {X 0,Y 321.079,Z 379.013,A -85,B 0,C 180,E1 -15592.713,E2 -15592.713} C_VEL
LIN {X 0,Y 315.677,Z 340.259,A -85,B 0,C 180,E1 -15593.975,E2 -15593.975} C_VEL
LIN {X 0,Y 316.055,Z 335.079,A -85,B 0,C 180,E1 -15595.345,E2 -15595.345} C_VEL
LIN {X 0,Y 314.482,Z 325.77,A -85,B 0,C 180,E1 -15597.99,E2 -15597.99} C_VEL
LIN {X 0,Y 312.56,Z 316.553,A -85,B 0,C 180,E1 -15600.768,E2 -15600.768} C_VEL
LIN {X 0,Y 312.511,Z 316.558,A -85,B 0,C 180,E1 -15604.211,E2 -15604.211} C_VEL
LIN {X 0,Y 312.515,Z 316.555,A -85,B 0,C 180,E1 -15607.388,E2 -15607.388} C_VEL
LIN {X 0,Y 312.445,Z 316.564,A -85,B 0,C 180,E1 -15610.717,E2 -15610.717} C_VEL
LIN {X 0,Y 312.456,Z 316.566,A -85,B 0,C 180,E1 -15614.21,E2 -15614.21} C_VEL
LIN {X 0,Y 312.488,Z 316.559,A -85,B 0,C 180,E1 -15617.919,E2 -15617.919} C_VEL
LIN {X 0,Y 312.502,Z 316.557,A -85,B 0,C 180,E1 -15620.971,E2 -15620.971} C_VEL
LIN {X 0,Y 312.537,Z 316.552,A -85,B 0,C 180,E1 -15624.221,E2 -15624.221} C_VEL
LIN {X 0,Y 312.506,Z 316.556,A -85,B 0,C 180,E1 -15627.334,E2 -15627.334} C_VEL
LIN {X 0,Y 312.529,Z 316.555,A -85,B 0,C 180,E1 -15631.286,E2 -15631.286} C_VEL
LIN {X 0,Y 312.559,Z 316.55,A -85,B 0,C 180,E1 -15634.708,E2 -15634.708} C_VEL
LIN {X 0,Y 312.569,Z 316.548,A -85,B 0,C 180,E1 -15637.527,E2 -15637.527} C_VEL
LIN {X 0,Y 312.571,Z 316.548,A -85,B 0,C 180,E1 -15641.652,E2 -15641.652} C_VEL
LIN {X 0,Y 312.69,Z 316.536,A -85,B 0,C 180,E1 -15645.686,E2 -15645.686} C_VEL
LIN {X 0,Y 312.702,Z 316.531,A -85,B 0,C 180,E1 -15649.642,E2 -15649.642} C_VEL
LIN {X 0,Y 312.834,Z 316.513,A -85,B 0,C 180,E1 -15652.253,E2 -15652.253} C_VEL
LIN {X 0,Y 312.705,Z 316.529,A -85,B 0,C 180,E1 -15654.842,E2 -15654.842} C_VEL
LIN {X 0,Y 312.987,Z 316.494,A -85,B 0,C 180,E1 -15658.713,E2 -15658.713} C_VEL
LIN {X 0,Y 312.987,Z 316.49,A -85,B 0,C 180,E1 -15661.286,E2 -15661.286} C_VEL
LIN {X 0,Y 312.701,Z 316.528,A -85,B 0,C 180,E1 -15665.158,E2 -15665.158} C_VEL
LIN {X 0,Y 312.8,Z 316.518,A -85,B 0,C 180,E1 -15667.747,E2 -15667.747} C_VEL
LIN {X 0,Y 312.668,Z 316.533,A -85,B 0,C 180,E1 -15671.671,E2 -15671.671} C_VEL
LIN {X 0,Y 312.671,Z 316.532,A -85,B 0,C 180,E1 -15674.864,E2 -15674.864} C_VEL
LIN {X 0,Y 312.552,Z 316.551,A -85,B 0,C 180,E1 -15679.193,E2 -15679.193} C_VEL
LIN {X 0,Y 312.529,Z 316.555,A -85,B 0,C 180,E1 -15682.779,E2 -15682.779} C_VEL
LIN {X 0,Y 312.541,Z 316.546,A -85,B 0,C 180,E1 -15685.91,E2 -15685.91} C_VEL
LIN {X 0,Y 312.506,Z 316.554,A -85,B 0,C 180,E1 -15689.654,E2 -15689.654} C_VEL
LIN {X 0,Y 312.522,Z 316.554,A -85,B 0,C 180,E1 -15693.688,E2 -15693.688} C_VEL
LIN {X 0,Y 312.523,Z 316.554,A -85,B 0,C 180,E1 -15697.385,E2 -15697.385} C_VEL
LIN {X 0,Y 312.492,Z 316.554,A -85,B 0,C 180,E1 -15700.709,E2 -15700.709} C_VEL
LIN {X 0,Y 312.454,Z 316.562,A -85,B 0,C 180,E1 -15704.209,E2 -15704.209} C_VEL
LIN {X 0,Y 312.485,Z 316.559,A -85,B 0,C 180,E1 -15707.918,E2 -15707.918} C_VEL
LIN {X 0,Y 312.479,Z 316.558,A -85,B 0,C 180,E1 -15710.967,E2 -15710.967} C_VEL
LIN {X 0,Y 312.533,Z 316.554,A -85,B 0,C 180,E1 -15714.219,E2 -15714.219} C_VEL
LIN {X 0,Y 312.504,Z 316.555,A -85,B 0,C 180,E1 -15717.333,E2 -15717.333} C_VEL
LIN {X 0,Y 312.526,Z 316.552,A -85,B 0,C 180,E1 -15721.285,E2 -15721.285} C_VEL
LIN {X 0,Y 312.556,Z 316.553,A -85,B 0,C 180,E1 -15724.707,E2 -15724.707} C_VEL
LIN {X 0,Y 312.589,Z 316.545,A -85,B 0,C 180,E1 -15727.528,E2 -15727.528} C_VEL
LIN {X 0,Y 312.59,Z 316.545,A -85,B 0,C 180,E1 -15731.652,E2 -15731.652} C_VEL
LIN {X 0,Y 312.686,Z 316.534,A -85,B 0,C 180,E1 -15735.685,E2 -15735.685} C_VEL
LIN {X 0,Y 312.676,Z 316.615,A -85,B 0,C 180,E1 -15737.67,E2 -15737.67} C_VEL
LIN {X 0,Y 314.191,Z 324.163,A -85,B 0,C 180,E1 -15740.01,E2 -15740.01} C_VEL
LIN {X 0,Y 318.179,Z 336.366,A -85,B 0,C 180,E1 -15740.565,E2 -15740.565} C_VEL
LIN {X 0,Y 321.581,Z 355.266,A -85,B 0,C 180,E1 -15741.221,E2 -15741.221} C_VEL
LIN {X 0,Y 319.882,Z 431.703,A -85,B 0,C 180,E1 -15742.94,E2 -15742.94} C_VEL
LIN {X 0,Y 319.325,Z 444.066,A -85,B 0,C 180,E1 -15743.443,E2 -15743.443} C_VEL
LIN {X 0,Y 318.541,Z 456.898,A -85,B 0,C 180,E1 -15744.222,E2 -15744.222} C_VEL
LIN {X 0,Y 317.541,Z 469.354,A -85,B 0,C 180,E1 -15745.261,E2 -15745.261} C_VEL
LIN {X 0,Y 316.414,Z 480.691,A -85,B 0,C 180,E1 -15746.497,E2 -15746.497} C_VEL
LIN {X 0,Y 315.179,Z 491.127,A -85,B 0,C 180,E1 -15747.922,E2 -15747.922} C_VEL
LIN {X 0,Y 314.154,Z 499.647,A -85,B 0,C 180,E1 -15749.358,E2 -15749.358} C_VEL
LIN {X 0,Y 313.183,Z 507.503,A -85,B 0,C 180,E1 -15750.963,E2 -15750.963} C_VEL
LIN {X 0,Y 312.299,Z 515.164,A -85,B 0,C 180,E1 -15752.901,E2 -15752.901} C_VEL
LIN {X 0,Y 311.643,Z 520.423,A -85,B 0,C 180,E1 -15754.526,E2 -15754.526} C_VEL
LIN {X 0,Y 311.279,Z 525.699,A -85,B 0,C 180,E1 -15756.576,E2 -15756.576} C_VEL
LIN {X 0,Y 310.925,Z 529.435,A -85,B 0,C 180,E1 -15758.447,E2 -15758.447} C_VEL
LIN {X 0,Y 310.633,Z 532.343,A -85,B 0,C 180,E1 -15760.427,E2 -15760.427} C_VEL
LIN {X 0,Y 310.582,Z 533.713,A -85,B 0,C 180,E1 -15761.75,E2 -15761.75} C_VEL
LIN {X 0,Y 310.555,Z 534.83,A -85,B 0,C 180,E1 -15763.319,E2 -15763.319} C_VEL
LIN {X 0,Y 310.537,Z 535.361,A -85,B 0,C 180,E1 -15765.757,E2 -15765.757} C_VEL
LIN {X 0,Y 310.844,Z 534.471,A -85,B 0,C 180,E1 -15768.27,E2 -15768.27} C_VEL
LIN {X 0,Y 311.081,Z 533.209,A -85,B 0,C 180,E1 -15769.807,E2 -15769.807} C_VEL
